DATA_BLOCK "Asi_output"	// DB 81
VERSION : 0.1
  STRUCT
   Adres_1_bit_0 : BOOL ;	//Temporary placeholder variable
   Adres_1_bit_1 : BOOL ;
   Adres_1_bit_2 : BOOL ;
   Adres_1_bit_3 : BOOL ;
   Adres_0_bit_0 : BOOL ;	//Temporary placeholder variable
   Adres_0_bit_1 : BOOL ;
   Adres_0_bit_2 : BOOL ;
   Adres_0_bit_3 : BOOL ;
   Adres_3_bit_0 : BOOL ;	//Temporary placeholder variable
   Adres_3_bit_1 : BOOL ;
   Adres_3_bit_2 : BOOL ;
   Adres_3_bit_3 : BOOL ;
   Adres_2_bit_0 : BOOL ;	//Temporary placeholder variable
   Adres_2_bit_1 : BOOL ;
   Adres_2_bit_2 : BOOL ;
   Adres_2_bit_3 : BOOL ;
   Adres_5_bit_0 : BOOL ;	//Temporary placeholder variable
   Adres_5_bit_1 : BOOL ;
   Adres_5_bit_2 : BOOL ;
   Adres_5_bit_3 : BOOL ;
   Adres_4_bit_0 : BOOL ;	//Temporary placeholder variable
   Adres_4_bit_1 : BOOL ;
   Adres_4_bit_2 : BOOL ;
   Adres_4_bit_3 : BOOL ;
   Adres_7_bit_0 : BOOL ;	//Temporary placeholder variable
   Adres_7_bit_1 : BOOL ;
   Adres_7_bit_2 : BOOL ;
   Adres_7_bit_3 : BOOL ;
   Adres_6_bit_0 : BOOL ;	//Temporary placeholder variable
   Adres_6_bit_1 : BOOL ;
   Adres_6_bit_2 : BOOL ;
   Adres_6_bit_3 : BOOL ;
   Adres_9_bit_0 : BOOL ;	//Temporary placeholder variable
   Adres_9_bit_1 : BOOL ;
   Adres_9_bit_2 : BOOL ;
   Adres_9_bit_3 : BOOL ;
   Adres_8_bit_0 : BOOL ;	//Temporary placeholder variable
   Adres_8_bit_1 : BOOL ;
   Adres_8_bit_2 : BOOL ;
   Adres_8_bit_3 : BOOL ;
   Adres_11_bit_0 : BOOL ;	//Temporary placeholder variable
   Adres_11_bit_1 : BOOL ;
   Adres_11_bit_2 : BOOL ;
   Adres_11_bit_3 : BOOL ;
   Adres_10_bit_0 : BOOL ;	//Temporary placeholder variable
   Adres_10_bit_1 : BOOL ;
   Adres_10_bit_2 : BOOL ;
   Adres_10_bit_3 : BOOL ;
   Adres_13_bit_0 : BOOL ;	//Temporary placeholder variable
   Adres_13_bit_1 : BOOL ;
   Adres_13_bit_2 : BOOL ;
   Adres_13_bit_3 : BOOL ;
   Adres_12_bit_0 : BOOL ;	//Temporary placeholder variable
   Adres_12_bit_1 : BOOL ;
   Adres_12_bit_2 : BOOL ;
   Adres_12_bit_3 : BOOL ;
   Adres_15_bit_0 : BOOL ;	//Temporary placeholder variable
   Adres_15_bit_1 : BOOL ;
   Adres_15_bit_2 : BOOL ;
   Adres_15_bit_3 : BOOL ;
   Adres_14_bit_0 : BOOL ;	//Temporary placeholder variable
   Adres_14_bit_1 : BOOL ;
   Adres_14_bit_2 : BOOL ;
   Adres_14_bit_3 : BOOL ;
   Adres_17_bit_0 : BOOL ;	//Temporary placeholder variable
   Adres_17_bit_1 : BOOL ;
   Adres_17_bit_2 : BOOL ;
   Adres_17_bit_3 : BOOL ;
   Adres_16_bit_0 : BOOL ;	//Temporary placeholder variable
   Adres_16_bit_1 : BOOL ;
   Adres_16_bit_2 : BOOL ;
   Adres_16_bit_3 : BOOL ;
   Adres_19_bit_0 : BOOL ;	//Temporary placeholder variable
   Adres_19_bit_1 : BOOL ;
   Adres_19_bit_2 : BOOL ;
   Adres_19_bit_3 : BOOL ;
   Adres_18_bit_0 : BOOL ;	//Temporary placeholder variable
   Adres_18_bit_1 : BOOL ;
   Adres_18_bit_2 : BOOL ;
   Adres_18_bit_3 : BOOL ;
   Adres_21_bit_0 : BOOL ;	//Temporary placeholder variable
   Adres_21_bit_1 : BOOL ;
   Adres_21_bit_2 : BOOL ;
   Adres_21_bit_3 : BOOL ;
   Adres_20_bit_0 : BOOL ;	//Temporary placeholder variable
   Adres_20_bit_1 : BOOL ;
   Adres_20_bit_2 : BOOL ;
   Adres_20_bit_3 : BOOL ;
   Adres_23_bit_0 : BOOL ;	//Temporary placeholder variable
   Adres_23_bit_1 : BOOL ;
   Adres_23_bit_2 : BOOL ;
   Adres_23_bit_3 : BOOL ;
   Adres_22_bit_0 : BOOL ;	//Temporary placeholder variable
   Adres_22_bit_1 : BOOL ;
   Adres_22_bit_2 : BOOL ;
   Adres_22_bit_3 : BOOL ;
   Adres_25_bit_0 : BOOL ;	//Temporary placeholder variable
   Adres_25_bit_1 : BOOL ;
   Adres_25_bit_2 : BOOL ;
   Adres_25_bit_3 : BOOL ;
   Adres_24_bit_0 : BOOL ;	//Temporary placeholder variable
   Adres_24_bit_1 : BOOL ;
   Adres_24_bit_2 : BOOL ;
   Adres_24_bit_3 : BOOL ;
   Adres_27_bit_0 : BOOL ;	//Temporary placeholder variable
   Adres_27_bit_1 : BOOL ;
   Adres_27_bit_2 : BOOL ;
   Adres_27_bit_3 : BOOL ;
   Adres_26_bit_0 : BOOL ;	//Temporary placeholder variable
   Adres_26_bit_1 : BOOL ;
   Adres_26_bit_2 : BOOL ;
   Adres_26_bit_3 : BOOL ;
   Adres_29_bit_0 : BOOL ;	//Temporary placeholder variable
   Adres_29_bit_1 : BOOL ;
   Adres_29_bit_2 : BOOL ;
   Adres_29_bit_3 : BOOL ;
   Adres_28_bit_0 : BOOL ;	//Temporary placeholder variable
   Adres_28_bit_1 : BOOL ;
   Adres_28_bit_2 : BOOL ;
   Adres_28_bit_3 : BOOL ;
   Adres_31_bit_0 : BOOL ;	//Temporary placeholder variable
   Adres_31_bit_1 : BOOL ;
   Adres_31_bit_2 : BOOL ;
   Adres_31_bit_3 : BOOL ;
   Adres_30_bit_0 : BOOL ;	//Temporary placeholder variable
   Adres_30_bit_1 : BOOL ;
   Adres_30_bit_2 : BOOL ;
   Adres_30_bit_3 : BOOL ;
   B_Adres_1_bit_0 : BOOL ;	//Temporary placeholder variable
   B_Adres_1_bit_1 : BOOL ;
   B_Adres_1_bit_2 : BOOL ;
   B_Adres_1_bit_3 : BOOL ;
   B_Adres_0_bit_0 : BOOL ;
   B_Adres_0_bit_1 : BOOL ;
   B_Adres_0_bit_2 : BOOL ;
   B_Adres_0_bit_3 : BOOL ;
   B_Adres_3_bit_0 : BOOL ;	//Temporary placeholder variable
   B_Adres_3_bit_1 : BOOL ;
   B_Adres_3_bit_2 : BOOL ;
   B_Adres_3_bit_3 : BOOL ;
   B_Adres_2_bit_0 : BOOL ;	//Temporary placeholder variable
   B_Adres_2_bit_1 : BOOL ;
   B_Adres_2_bit_2 : BOOL ;
   B_Adres_2_bit_3 : BOOL ;
   B_Adres_5_bit_0 : BOOL ;	//Temporary placeholder variable
   B_Adres_5_bit_1 : BOOL ;
   B_Adres_5_bit_2 : BOOL ;
   B_Adres_5_bit_3 : BOOL ;
   B_Adres_4_bit_0 : BOOL ;	//Temporary placeholder variable
   B_Adres_4_bit_1 : BOOL ;
   B_Adres_4_bit_2 : BOOL ;
   B_Adres_4_bit_3 : BOOL ;
   B_Adres_7_bit_0 : BOOL ;	//Temporary placeholder variable
   B_Adres_7_bit_1 : BOOL ;
   B_Adres_7_bit_2 : BOOL ;
   B_Adres_7_bit_3 : BOOL ;
   B_Adres_6_bit_0 : BOOL ;	//Temporary placeholder variable
   B_Adres_6_bit_1 : BOOL ;
   B_Adres_6_bit_2 : BOOL ;
   B_Adres_6_bit_3 : BOOL ;
   B_Adres_9_bit_0 : BOOL ;	//Temporary placeholder variable
   B_Adres_9_bit_1 : BOOL ;
   B_Adres_9_bit_2 : BOOL ;
   B_Adres_9_bit_3 : BOOL ;
   B_Adres_8_bit_0 : BOOL ;	//Temporary placeholder variable
   B_Adres_8_bit_1 : BOOL ;
   B_Adres_8_bit_2 : BOOL ;
   B_Adres_8_bit_3 : BOOL ;
   B_Adres_11_bit_0 : BOOL ;	//Temporary placeholder variable
   B_Adres_11_bit_1 : BOOL ;
   B_Adres_11_bit_2 : BOOL ;
   B_Adres_11_bit_3 : BOOL ;
   B_Adres_10_bit_0 : BOOL ;	//Temporary placeholder variable
   B_Adres_10_bit_1 : BOOL ;
   B_Adres_10_bit_2 : BOOL ;
   B_Adres_10_bit_3 : BOOL ;
   B_Adres_13_bit_0 : BOOL ;	//Temporary placeholder variable
   B_Adres_13_bit_1 : BOOL ;
   B_Adres_13_bit_2 : BOOL ;
   B_Adres_13_bit_3 : BOOL ;
   B_Adres_12_bit_0 : BOOL ;	//Temporary placeholder variable
   B_Adres_12_bit_1 : BOOL ;
   B_Adres_12_bit_2 : BOOL ;
   B_Adres_12_bit_3 : BOOL ;
   B_Adres_15_bit_0 : BOOL ;	//Temporary placeholder variable
   B_Adres_15_bit_1 : BOOL ;
   B_Adres_15_bit_2 : BOOL ;
   B_Adres_15_bit_3 : BOOL ;
   B_Adres_14_bit_0 : BOOL ;	//Temporary placeholder variable
   B_Adres_14_bit_1 : BOOL ;
   B_Adres_14_bit_2 : BOOL ;
   B_Adres_14_bit_3 : BOOL ;
   B_Adres_17_bit_0 : BOOL ;	//Temporary placeholder variable
   B_Adres_17_bit_1 : BOOL ;
   B_Adres_17_bit_2 : BOOL ;
   B_Adres_17_bit_3 : BOOL ;
   B_Adres_16_bit_0 : BOOL ;	//Temporary placeholder variable
   B_Adres_16_bit_1 : BOOL ;
   B_Adres_16_bit_2 : BOOL ;
   B_Adres_16_bit_3 : BOOL ;
   B_Adres_19_bit_0 : BOOL ;	//Temporary placeholder variable
   B_Adres_19_bit_1 : BOOL ;
   B_Adres_19_bit_2 : BOOL ;
   B_Adres_19_bit_3 : BOOL ;
   B_Adres_18_bit_0 : BOOL ;	//Temporary placeholder variable
   B_Adres_18_bit_1 : BOOL ;
   B_Adres_18_bit_2 : BOOL ;
   B_Adres_18_bit_3 : BOOL ;
   B_Adres_21_bit_0 : BOOL ;	//Temporary placeholder variable
   B_Adres_21_bit_1 : BOOL ;
   B_Adres_21_bit_2 : BOOL ;
   B_Adres_21_bit_3 : BOOL ;
   B_Adres_20_bit_0 : BOOL ;	//Temporary placeholder variable
   B_Adres_20_bit_1 : BOOL ;
   B_Adres_20_bit_2 : BOOL ;
   B_Adres_20_bit_3 : BOOL ;
   B_Adres_23_bit_0 : BOOL ;	//Temporary placeholder variable
   B_Adres_23_bit_1 : BOOL ;
   B_Adres_23_bit_2 : BOOL ;
   B_Adres_23_bit_3 : BOOL ;
   B_Adres_22_bit_0 : BOOL ;	//Temporary placeholder variable
   B_Adres_22_bit_1 : BOOL ;
   B_Adres_22_bit_2 : BOOL ;
   B_Adres_22_bit_3 : BOOL ;
   B_Adres_25_bit_0 : BOOL ;	//Temporary placeholder variable
   B_Adres_25_bit_1 : BOOL ;
   B_Adres_25_bit_2 : BOOL ;
   B_Adres_25_bit_3 : BOOL ;
   B_Adres_24_bit_0 : BOOL ;	//Temporary placeholder variable
   B_Adres_24_bit_1 : BOOL ;
   B_Adres_24_bit_2 : BOOL ;
   B_Adres_24_bit_3 : BOOL ;
   B_Adres_27_bit_0 : BOOL ;	//Temporary placeholder variable
   B_Adres_27_bit_1 : BOOL ;
   B_Adres_27_bit_2 : BOOL ;
   B_Adres_27_bit_3 : BOOL ;
   B_Adres_26_bit_0 : BOOL ;	//Temporary placeholder variable
   B_Adres_26_bit_1 : BOOL ;
   B_Adres_26_bit_2 : BOOL ;
   B_Adres_26_bit_3 : BOOL ;
   B_Adres_29_bit_0 : BOOL ;	//Temporary placeholder variable
   B_Adres_29_bit_1 : BOOL ;
   B_Adres_29_bit_2 : BOOL ;
   B_Adres_29_bit_3 : BOOL ;
   B_Adres_28_bit_0 : BOOL ;	//Temporary placeholder variable
   B_Adres_28_bit_1 : BOOL ;
   B_Adres_28_bit_2 : BOOL ;
   B_Adres_28_bit_3 : BOOL ;
   B_Adres_31_bit_0 : BOOL ;	//Temporary placeholder variable
   B_Adres_31_bit_1 : BOOL ;
   B_Adres_31_bit_2 : BOOL ;
   B_Adres_31_bit_3 : BOOL ;
   B_Adres_30_bit_0 : BOOL ;	//Temporary placeholder variable
   B_Adres_30_bit_1 : BOOL ;
   B_Adres_30_bit_2 : BOOL ;
   B_Adres_30_bit_3 : BOOL ;
  END_STRUCT ;	
BEGIN
END_DATA_BLOCK

DATA_BLOCK "MPI_GD"	// DB 100
VERSION : 0.1
  STRUCT
   IN : STRUCT
    Life_Bit_Foliarka : BOOL ;
    Foliarka_Automatyka : BOOL ;
    Foliarka_Reczny : BOOL ;
    Foto_Banda_1 : BOOL ;
    Foto_Owijarka : BOOL ;
    Rezerwa_1 : BOOL ;
    Motor_10_Lewo : BOOL ;
    Motor_10_Prawo : BOOL ;
    Motor_11_Lewo : BOOL ;
    Motor_11_Prawo : BOOL ;
    Zezwolenie_Na_Wjazd_10 : BOOL ;
    Potw_Dost_Na_Wjazd_10 : BOOL ;
    Zabierz_Na_Bande_11 : BOOL ;
    Paleta_Obecna_Na_7_Tr : BOOL ;
    Help_INT : INT ;
   END_STRUCT ;
   OUT : STRUCT
    Life_Bit_Szafa : BOOL ;
    Szafa_Automatyka : BOOL ;
    Foto_1_Banda_10 : BOOL ;
    Foto_2_Banda_10 : BOOL ;
    Foto_Banda_11 : BOOL ;
    Silnik_10_OK : BOOL ;
    Silnik_11_OK : BOOL ;
    Zabierz_Na_Bande_10 : BOOL ;
    Zezwolenie_Na_Wyjazd_11 : BOOL ;
    Potw_Dost_Na_Wyjazd_11 : BOOL ;
    Obrot_Na_Poz_Wlot_1 : BOOL ;
    Zmien_Program_Na_4 : BOOL ;
    Zmien_Pragram_Na_3 : BOOL ;
    Foto_Banda_9 : BOOL ;
    Help_INT : INT ;
   END_STRUCT ;
  END_STRUCT ;	
BEGIN
END_DATA_BLOCK

DATA_BLOCK "Blok_Bledow"	// DB 119
VERSION : 0.1
  STRUCT
   Blad_Silnika_Adr_1 : BOOL ;	//Blad silnika o adresie 1 - rolki obrotnica bindownicy
   Blad_Silnika_Adr_2 : BOOL ;	//Blad silnika o adresie 2 - rolki wylot bindownicy
   Blad_Silnika_Adr_3 : BOOL ;	//Blad silnika o adresie 3 - rolki
   Blad_Silnika_Adr_4 : BOOL ;	//Blad silnika o adresie 4 - rolki
   Blad_Silnika_Adr_5 : BOOL ;	//Blad silnika o adresie 5 - rolki
   Blad_Silnika_Adr_6 : BOOL ;	//Blad silnika o adresie 6 - rolki
   Blad_Silnika_Adr_7 : BOOL ;	//Blad silnika o adresie 7 - rolki
   Blad_Silnika_Adr_8 : BOOL ;	//Blad silnika o adresie 8 - rolki
   Blad_Silnika_Adr_9 : BOOL ;	//Blad silnika o adresie 9 - rolki
   Blad_Silnika_Adr_10 : BOOL ;	//Blad silnika o adresie 10 - rolki
   Blad_Silnika_Adr_11 : BOOL ;	//Blad silnika o adresie 11 - rolki
   Blad_Silnika_Adr_12 : BOOL ;	//Blad silnika o adresie 12 - rolki
   Blad_Silnika_Adr_13 : BOOL ;	//Blad silnika o adresie 13 - rolki
   Blad_Silnika_Adr_14 : BOOL ;	//Blad silnika o adresie 14 - rolki
   Blad_Silnika_Adr_15 : BOOL ;	//Blad silnika o adresie 15 - silnik obrotnicy bindownicy
   Blad_Rygla_Adr_16 : BOOL ;	//Blad rygla drzwi o adresie 16
   Blad_Silnika_Adr_18 : BOOL ;	//Blad silnika o adresie 18 - silnik obrotnicy wyboru wlotu
   Blad_Silnika_Adr_20 : BOOL ;	//Blad silnika o adresie 20 - silnik obrotnicy etykietownicy
   Blad_Silnika_Adr_23 : BOOL ;	//Blad silnika o adresie 23 - rolki
   Blad_Silnika_Adr_24 : BOOL ;	//Blad silnika o adresie 24 - rolki
   Blad_Kurtyny_Adr_25 : BOOL ;	//Blad kurtyny wlotowej  adres 25
   Blad_Kurtyny_Adr_26 : BOOL ;	//Blad kurtyny wylotowej aders 26
   Blad_Not_Aus_27 : BOOL ;	//Blad Not Aus adres 27 - Not Aus szafa
   Blad_Not_Aus_28 : BOOL ;	//Blad Not Aus adres 28 - Not Aus poczatek lini
   Blad_Not_Aus_29 : BOOL ;	//Blad Not Aus adres 29 - Not Aus srodek lini
   Blad_Not_Aus_30 : BOOL ;	//Blad Not Aus adres 30 - Not Aus koniec lini
   Blad_Not_Aus_31 : BOOL ;	//Blad Not Aus adres 31 - Not Aus panel bindownicy
   Blad_Przek_Bezp_Bind : BOOL ;	//Strefa bezpieczenstwa rejonu bindownicy  niepotwierdzona(wejscie -I4.4)
   Ostrz_Bind_Blad : BOOL ;	//Blad ogolny bindownicy
   Ostrz_Bind_Nie_Cofnieta : BOOL ;	//Bindownica nie jest cofnieta
   Ostrz_Bind_Sygn_Bezp : BOOL ;	//Bindownica brak sygnalu bezpieczenstwa
   Ostrz_Bind_Nie_Jest_Auto : BOOL ;	//Bindownica nie jest w trybie automatycznym (wejscie -I2.4)
   Ostrz_Stol_Obr_Foto : BOOL ;	//Blad fotokomorek stolu obrotowego
   Ostrz_Obr_Stol_Obr_Pozyc : BOOL ;	//Stol obrotowy nie jest w pozycji 0
   Ostrz_Pokr_Foto_Tas_1 : BOOL ;	//Niewlasciwe Pokrycie fotkomorek na tasmie 1 (Przejedz do przodu w recznym )
   Ostrz_Pokr_Foto_Tas_2 : BOOL ;	//Niewlasciwe Pokrycie fotkomorek na tasmie 2 (Przejedz do przodu w recznym )
   Ostrz_Pokr_Foto_Obr : BOOL ;	//Niewlasciwe Pokrycie fotkomorek na obrotnicy (Przejedz do przodu w recznym )
   Ostrz_Pokr_Foto_Tas_4 : BOOL ;	//Niewlasciwe Pokrycie fotkomorek na tasmie 4 (Przejedz do przodu w recznym )
   Blad_Krok_1 : BOOL ;	//Blad kroku nr 1 (Przekrokczony czas jazdy  na zadana pozycje)
   Blad_Krok_2 : BOOL ;	//Blad kroku nr 2 (Przekrokczony czas szukania srodka palety)
   Blad_Krok_3 : BOOL ;	//Blad kroku nr 3 (Przekrokczony czas pozycjonowania palety lewo/prawo)
   Blad_Krok_4 : BOOL ;	//Blad kroku nr 4 (Przekrokczony czas strzalu bindownicy)
   Blad_Krok_5 : BOOL ;	//Blad kroku nr 5 (Przekrokczony czas czasu postoju)
   Blad_Krok_6 : BOOL ;	//Blad kroku nr 6 (Przekrokczony czas powrotu lewo/prawo)
   Alarm_Obr_Stol_Obr_Pozyc : BOOL ;	//Stol obrotowy nie jest w pozycji 0
   Alarm_Bind_Nie_Cofinieta : BOOL ;	//Bindownica nie cofnieta lub brak zezwolenia  (cofnij ramie do tylu)
   Alarm_Bind_Sygn_Bezp : BOOL ;	//Bindownica brak sygnalu bezpieczenstwa
   rez3 : BOOL ;	//rez 3
   rez_6_0 : BOOL ;	//rez_6_0
   Alarm_Pokr_Foto_Tas_1 : BOOL ;	//Niewlasciwe Pokrycie fotkomorek na tasmie 1 (Przejedz do przodu w recznym )
   Alarm_Pokr_Foto_Tas_2 : BOOL ;	//Niewlasciwe Pokrycie fotkomorek na tasmie 2 (Przejedz do przodu w recznym )
   Alarm_Pokr_Foto_Tas_4 : BOOL ;	//Niewlasciwe Pokrycie fotkomorek na tasmie 4 (Przejedz do przodu w recznym )
   Alarm_Pokr_Foto_Obr : BOOL ;	//Niewlasciwe Pokrycie fotkomorek na obrotnicy przy braku cyklu
   Alarm_Bind_Nie_Jest_Auto : BOOL ;	//Bindownica nie jest w trybie automatycznym (wejscie -I2.4)
   Alarm_Bind_Blad : BOOL ;	//Blad ogolny bindownicy
   rez_6_7 : BOOL ;	//rez_6_7
   Ostrz_Prasa_Nie_W_Gorze : BOOL ;	//Zlamywak dekli nie jest u gory I2.6
   rez_7_1 : BOOL ;	//rez_7_1
   rez_7_2 : BOOL ;	//rez_7_2
   rez_7_3 : BOOL ;	//rez_7_3
   rez_7_4 : BOOL ;	//rez_7_4
   rez_7_5 : BOOL ;	//rez_7_5
   Ostrz_Wozek_Przy_Przen : BOOL ;	//Wozek widlowy przy przenosniku (i2.7)
   Ostrz_C_Bind_Foto_Pokr : BOOL ;	//Pokrycie fotokomorek podczas cyklu bindowania
   Ostrz_C_Bind_Poz_Bindow : BOOL ;	//Pozycja bindownicy podczas bindowania
   rez_8_1 : BOOL ;	//rez_8_1
   rez_8_2 : BOOL ;	//rez_8_2
   rez_8_3 : BOOL ;	//rez_8_3
   rez_8_4 : BOOL ;	//rez_8_4
   rez_8_5 : BOOL ;	//rez_8_5
   rez_8_6 : BOOL ;	//rez_8_6
   rez_8_7 : BOOL ;	//rez_8_7
   rez_9_0 : BOOL ;	//rez_9_0
   rez_9_1 : BOOL ;	//rez_9_1
   rez_9_2 : BOOL ;	//rez_9_2
   rez_9_3 : BOOL ;	//rez_9_3
   rez_9_4 : BOOL ;	//rez_9_4
   rez_9_5 : BOOL ;	//rez_9_5
   rez_9_6 : BOOL ;	//rez_9_6
   rez_9_7 : BOOL ;	//rez_9_7
   rez_int_bl : INT ;
   rez_int_bl_2 : INT ;
  END_STRUCT ;	
BEGIN
END_DATA_BLOCK

DATA_BLOCK "DB_HMI"	// DB 120
VERSION : 0.1
  STRUCT
   HMI_IN : STRUCT 	//Zmienne wchodzace do HMI nie nadpisywane W HMI (100 bajtow)
    Tryb_Reczny : BOOL ;	//Tryb Reczny
    Tryb_Auto : BOOL ;	//Tryb Auto
    Pozycja_0_st : BOOL ;	//Obrotnica Pozycja 0 st
    Pozycja_90_st : BOOL ;	//Obrotnica Pozycja 90 st
    Pozycja_180_st : BOOL ;	//Obrotnica Pozycja 180 st
    Pozycja_270_st : BOOL ;	//Obrotnica Pozycja 270 st
    Foto_Tasma_1_Tyl : BOOL ;	//foto tylne na bandzie wlotowej
    Foto_Tasma_1_Przod : BOOL ;	//foto przednie bandzie wlotowej
    Foto_Tasma_2_Tyl : BOOL ;	//foto tylne na bandzie wlotowej 2
    Foto_Tasma_2_Przod : BOOL ;	//foto przednie na bandzie wlotowej 2
    Foto_Obrotnica_3_Tyl : BOOL ;	//foto tylne na obrotnicy 3
    Foto_Obrotnica_3_Przod : BOOL ;	//foto przednie na obrotnicy 3
    Foto_Tasma_4_Tyl : BOOL ;	//foto tylne na bandzie wylotowej 4
    Foto_Tasma_4_Przod : BOOL ;	//foto przednie na bandzie wlotowej 4
    Motor_Tasma_1_Tyl : BOOL ;	//motor tasma 1 tyl
    Motor_Tasma_1_Przod : BOOL ;	//motor tasma 1 przod
    Motor_Tasma_2_Tyl : BOOL ;	//motor tasma 2 tyl
    Motor_Tasma_2_Przod : BOOL ;	//motor tasma 2 przod
    Motor_Tasma_3_Tyl : BOOL ;	//motor tasma obrotnica 3 tyl
    Motor_Tasma_3_Przod : BOOL ;	//motor tasma obrotnica 3 przod
    Motor_Obrotnica_3_CW : BOOL ;	//motor obrotnica 3 clock wise
    Motor_Obrotnica_3_CCW : BOOL ;	//motor obrotnica 3 counter clock wise
    Motor_Tasma_4_Przod : BOOL ;	//motor tasma obrotnica 4 tyl
    Motor_Tasma_4_Tyl : BOOL ;	//motor tasma obrotnica 4 przod
    Kurtyna_Wlot_Ok : BOOL ;	//kurtyna na wlocie ok
    Kurtyna_Wylot_Ok : BOOL ;	//kurtyna na wylocie ok
    Wybrano_TP_Przelot : BOOL ;	//wybrano tryb pracy przelot
    Wybrano_TP_Wiazanie_Wzdl : BOOL ;	//wybrano tryb pracy wiazanie wzdluzne
    Wybrano_TP_Wiazanie_Pop : BOOL ;	//wybrano tryb pracy wiazanie poprzeczne
    Wybrano_TP_Wiazanie_Krzy : BOOL ;	//wybrano tryb pracy wiazanie krzyzowe
    Czujnik_Ham_0_St : BOOL ;	//fotokomorka hamowania obrotnicy do kata 0st
    Czujnik_0_St : BOOL ;	//fotokomorka zatrzymania obrotnicy przy kacie 0st
    Czujnik_Ham_90_St : BOOL ;	//fotokomorka hamowania obrotnicy do kata 90st
    Czujnik_90_St : BOOL ;	//fotokomorka zatrzymania obrotnicy przy kacie 90st
    Czujnik_Ham_180_St : BOOL ;	//fotokomorka hamowania obrotnicy do kata 180st
    Czujnik_180_St : BOOL ;	//fotokomorka zatrzymania obrotnicy przy kacie 180st
    Czujnik_Ham_270_St : BOOL ;	//fotokomorka hamowania obrotnicy do kata 270st
    Czujnik_270_St : BOOL ;	//fotokomorka zatrzymania obrotnicy przy kacie 270st
    Interfefs_B_do_TP_B1 : BOOL ;	//obwod bezpieczenstwa bindownicy
    Interfefs_B_do_TP_B2 : BOOL ;	//polozenie podstawowe bindownicy
    Interfefs_B_do_TP_B3 : BOOL ;	//start/zakonczenie wiazania
    Interfefs_B_do_TP_B5 : BOOL ;	//blad bindownicy
    Interfefs_TP_do_B_TP1 : BOOL ;	//obwod bezpieczenstwa tasmociagow
    Interfefs_TP_do_B_TP2 : BOOL ;	//zezwolenie na prace bindownicy
    Interfefs_TP_do_B_TP3 : BOOL ;	//start wiazania
    PB_Strefa_bezpieczenstwa : BOOL ;	//przycisk zalaczenie Strefy bezpieczenstwa
    PB_Reczny : BOOL ;	//przycisk trybu reczny
    PB_Auto : BOOL ;	//przycisk auto
    PB_Reset : BOOL ;	//przycisk reset
    PB_Stop : BOOL ;	//przycisk stop
    PB_Cykl_Start : BOOL ;	//przycisk start cyklu
    PB_Tasma1_Tyl : BOOL ;	//przycisk tasma 1 do tylu
    PB_Tasma1_Przod : BOOL ;	//przycisk tasma 1 do przodu
    PB_Tasma2_Tyl : BOOL ;	//przycisk tasma 2 do tylu
    PB_Tasma2_Przod : BOOL ;	//przycisk tasma 2 do przodu
    PB_Tasma3_Tyl : BOOL ;	//przycisk tasma 3 do tylu
    PB_Tasma3_Przod : BOOL ;	//przycisk tasma 3 do przodu
    PB_Tasma4_Tyl : BOOL ;	//przycisk tasma 4 do tylu
    PB_Tasma4_Przod : BOOL ;	//przycisk tasma 4 do przodu
    PB_Tasma3_Obr_CW : BOOL ;	//przycisk obrotnica w prawo
    PB_Tasma3_Obr_CCW : BOOL ;	//przycisk obrotnica w lewo
    Lampka_Blad_Bind : BOOL ;	//lamka bledu bindownicy
    Lampka_Strzal_Tasmy : BOOL ;	//lampka wystrzalu tasmy
    Lampka_Strefa_Bezp : BOOL ;	//lampka przycisku strefy bezpieczenstwa
    Lampka_PB_Reczny : BOOL ;	//lampka przycisku trybu recznego
    Lampka_PB_Auto : BOOL ;	//lampka przycisku trybu auto
    Lampka_PB_Reset : BOOL ;	//lampka przycisku reset
    Lampka_PB_Stop : BOOL ;	//lampka przycisku stop
    Lampka_PB_Cykl_Start : BOOL ;	//lampka przycisku start
    Paleta_na_Tasmie_1 : BOOL ;	//znacznik palety na tasmie 1
    Paleta_na_Tasmie_2 : BOOL ;	//znacznik palety na tasmie 2
    Paleta_na_Tasmie_3_0_180 : BOOL ;	//znacznik palety na tasmie 3 przy kacie 0 lub 180st
    Paleta_na_Tasmie_3_90_27 : BOOL ;	//znacznik palety na tasmie 3 przy kacie 90 lub 270st
    Paleta_na_Tasmie_4 : BOOL ;	//znacznik palety na tasmie 4
    Paleta_na_Tasmie_1_T : BOOL ;	//znacznik palety na tasmie 1 wjazd
    Paleta_na_Tasmie_1_P : BOOL ;	//znacznik palety na tasmie 1 wyjazd
    Paleta_na_Tasmie_2_T : BOOL ;	//znacznik palety na tasmie 2 wjazd
    Paleta_na_Tasmie_2_P : BOOL ;	//znacznik palety na tasmie 2 wyjazd
    Paleta_na_Tasmie_3_T : BOOL ;	//znacznik palety na tasmie 3 wjazd
    Paleta_na_Tasmie_3_P : BOOL ;	//znacznik palety na tasmie 3 wyjazd
    Paleta_na_Tasmie_4_T : BOOL ;	//znacznik palety na tasmie 4 wjazd
    Paleta_na_Tasmie_4_P : BOOL ;	//znacznik palety na tasmie 4 wyjazd
    Rygiel : BOOL ;	//znacznik rygla drzwi
    Blad : BOOL ;	//Znacznik bledu
    Linia_transportowa_praca : BOOL ;	//Znacznik pracy calej linii transportowej
    Interfefs_B_do_TP_B4 : BOOL ;	//tryb pracy bindownicy: Auto(1) Reczny(0)
    Krok_1 : BOOL ;	//krok 1 trybu pracy
    Krok_2 : BOOL ;	//krok 2 trybu pracy
    Krok_3 : BOOL ;	//krok 3 trybu pracy
    Krok_4 : BOOL ;	//krok 4 trybu pracy
    Krok_5 : BOOL ;	//krok 5 trybu pracy
    Krok_6 : BOOL ;	//krok 6 trybu pracy
    Znacznik_Migania_Bledu : BOOL ;	//znacznik migania bledu
    Czujnik_Prasa : BOOL ;	//czujnik prasy s 22
    Stan_Zaworu : BOOL ;
    Tablica_IN_bool : ARRAY  [1 .. 10 ] OF BOOL  := FALSE;
    Tablica_IN_Byte : ARRAY  [1 .. 6 ] OF BYTE  := B#16#0;
    input_0 : BYTE ;
    input_1 : BYTE ;
    input_2 : BYTE ;
    input_3 : BYTE ;
    output_0 : BYTE ;
    output_1 : BYTE ;
    output_2 : BYTE ;
    output_3 : BYTE ;
    input_8 : BYTE ;
    input_9 : BYTE ;
    input_10 : BYTE ;
    input_11 : BYTE ;
    Tablica_IN_DWORD : ARRAY  [1 .. 4 ] OF DWORD ;
    NR_Kroku : DINT ;	//Numer kroku
    Aktualna_Data : DATE_AND_TIME ;
    Tablica_IN_INT : ARRAY  [1 .. 18 ] OF INT ;
    tryb_wiaz : INT ;	//znacznik wyboru trybu wiazania
    INT_Liczba_Akt_Kroku : INT ;	//znacznik wyboru aktualnie wykonywanego kroku
   END_STRUCT ;
   HMI_OUT : STRUCT 	//Zmienne wychodzace z HMI Nie nadpisywane w sterowniku od 100 bajta
    Rezerwa_Out_1 : BOOL ;
    Rezerwa_Out_2 : BOOL ;
    Start_Lini_z_OP : BOOL ;	//start calej lini z HMI
    Stop_Lini_z_OP : BOOL ;	//stop calej lini z HMI
    Wyzwolenie_Wyjazdu : BOOL ;	//wyzwolenie wyjazdu palety na stanowisku bindujacym (tylko w auto)
    Przycisk_Test_Lampek : BOOL ;	//przycisk test lampek
    Przycisk_Reset_Bledow : BOOL ;	//Przycisk resetowania bledow na panelu HMI
    Przycisk_Pozycjonowanie : BOOL ;	//Przycisk HMI do pozycjonowania palety
    H_Zalacz_Zawor_Prasa : BOOL ;	//Zalacz zawor prasa
    H_Zezwl_Ekran_Prasa : BOOL ;	//Zezwolenie na prase reczny
    Tablica_OUT_Bool : ARRAY  [1 .. 144 ] OF BOOL ;
    Tablina_OUT_INT : ARRAY  [1 .. 40 ] OF INT ;
   END_STRUCT ;
   HMI_IN_OUT : STRUCT 	//Zmienne nadpisywane w sterowniku i w HMI od 200 bajta
    Rezerwa_IN_Out_1 : BOOL ;
    Tp_Przelot : BOOL ;	//Tryb Pracy Przelot
    Tp_Wiazanie_Poprzeczne : BOOL ;	//Tryb Pracy Wiazanie poprzeczne
    Tp_Wiazanie_Wzdluzne : BOOL ;	//Tryb Pracy Wiazanie wzduzne
    Tp_Wiazanie_Pop_Wzdl : BOOL ;	//Tryb Pracy Wiaznie Poprzeczne i wzdluzne
    Tp_Pozycjonowanie : BOOL ;	//Tryb Pracy Pozycjonowanie Palety zalaczone
    Test_Lampek : BOOL ;	//Test Lampek
    Reset_bledow : BOOL ;	//Reset Bledow
    Zlamywak_Dekl : BOOL ;	//lamanie dekli
    Tablica_IN_OUT_Bool : ARRAY  [1 .. 144 ] OF BOOL ;
    Tablica_IN_OUT_INT : ARRAY  [1 .. 40 ] OF INT ;
    Wybor_trybu_pracy : BYTE ;
   END_STRUCT ;
  END_STRUCT ;	
BEGIN
   HMI_IN.Foto_Obrotnica_3_Przod := TRUE;
END_DATA_BLOCK

DATA_BLOCK DB 200
VERSION : 0.1
  STRUCT
   Wiazanie_Wzdluzne : BOOL ;	//wiazanie wzdluz palety
   Wiazanie_Poprzeczne : BOOL ;	//wiaznaie w poprzek palety
   Czas_Kontr_Rolki_Wlot : TIME  := T#12S;	//czas kontrolny wlotu
   Czas_Dojazd_Rolki_Wlot : TIME  := T#100MS;	//czas dojazdu do fotokomorki
   Czas_Opoz_Opusz_Bandy : TIME  := T#2S;	//czas po ktorym paleta opuszcza bande
   Czas_Opusz_Bandy : TIME  := T#2S;
   Czas_Opoz_Po_Strzale : TIME  := T#2S;
   Pozycjonowanie : BOOL ;	//jezeli true paleta pozycjonowana
   Pozycj_0_Lewo : BOOL ;	//pozycjonowanie 0st
   Pozycj_0_Prawo : BOOL ;	//pozycjonowanie 0st
   Pozycj_180_Lewo : BOOL ;	//pozycjonowanie 180st
   Pozycjo_180_Prawo : BOOL ;	//pozycjonowanie 180st
   Pozycj_0_Lewo_Czas : TIME  := T#2S;	//pozycjonowanie w lewo czas
   Pozycj_0_Prawo_Czas : TIME  := T#2S;	//pozycjonowanie w prawo czas
   Pozycj_180_Lewo_Czas : TIME  := T#2S;	//pozycjonowanie w lewo czas
   Pozycj_180_Prawo_Czas : TIME  := T#2S;	//pozycjonowanie w lewo czas
  END_STRUCT ;	
BEGIN
   Czas_Kontr_Rolki_Wlot := T#12S;
   Czas_Dojazd_Rolki_Wlot := T#100MS;
   Czas_Opoz_Opusz_Bandy := T#2S;
   Czas_Opusz_Bandy := T#2S;
   Czas_Opoz_Po_Strzale := T#2S;
   Pozycj_0_Lewo_Czas := T#2S;
   Pozycj_0_Prawo_Czas := T#2S;
   Pozycj_180_Lewo_Czas := T#2S;
   Pozycj_180_Prawo_Czas := T#2S;
END_DATA_BLOCK

ORGANIZATION_BLOCK OB 1
TITLE = "Main Program Sweep (Cycle)"
VERSION : 0.1
VAR_TEMP
  OB1_EV_CLASS : BYTE ;	//Bits 0-3 = 1 (Coming event), Bits 4-7 = 1 (Event class 1)
  OB1_SCAN_1 : BYTE ;	//1 (Cold restart scan 1 of OB 1), 3 (Scan 2-n of OB 1)
  OB1_PRIORITY : BYTE ;	//Priority of OB Execution
  OB1_OB_NUMBR : BYTE ;	//1 (Organization block 1, OB1)
  OB1_RESERVED_1 : BYTE ;	//Reserved for system
  OB1_RESERVED_2 : BYTE ;	//Reserved for system
  OB1_PREV_CYCLE : INT ;	//Cycle time of previous OB1 scan (milliseconds)
  OB1_MIN_CYCLE : INT ;	//Minimum cycle time of OB1 (milliseconds)
  OB1_MAX_CYCLE : INT ;	//Maximum cycle time of OB1 (milliseconds)
  OB1_DATE_TIME : DATE_AND_TIME ;	//Date and time OB1 started
END_VAR
BEGIN
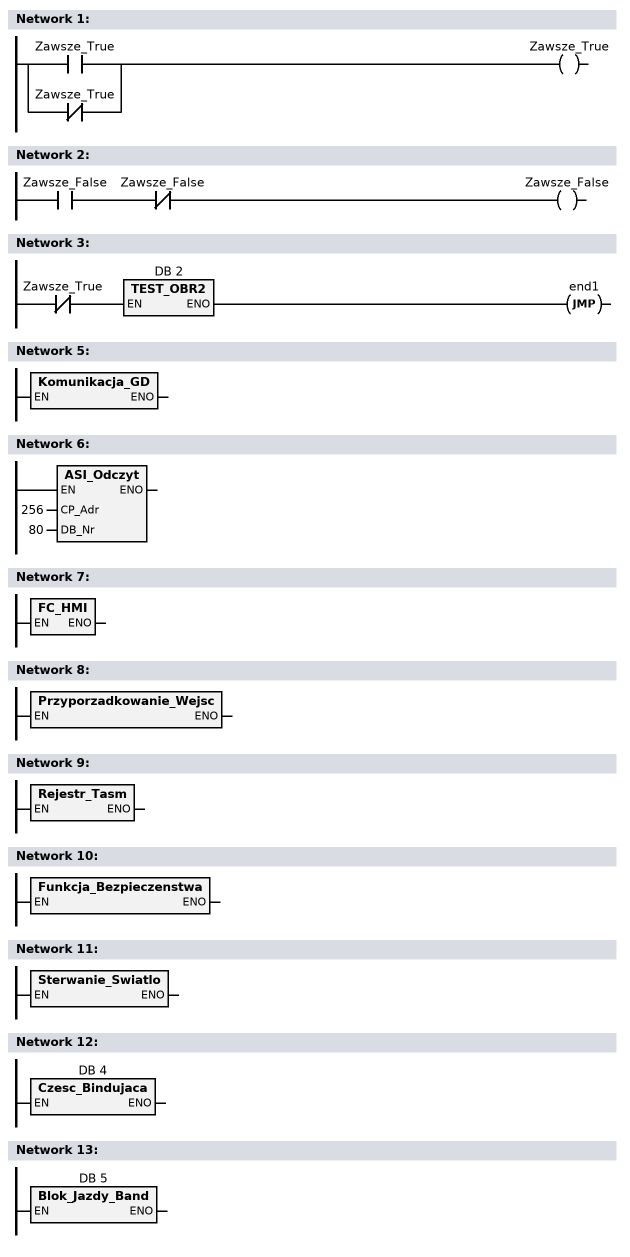
NETWORK
TITLE =
//Zawsze true
      O     "Zawsze_True";
      ON    "Zawsze_True";
      =     "Zawsze_True";
NETWORK
TITLE =
//Zawsze False
      A     "Zawsze_False";
      AN    "Zawsze_False";
      =     "Zawsze_False";
NETWORK
TITLE =
//Nie uzywany w normalej pracy blok
      AN    "Zawsze_True";
      JNB   _001;
      CALL  "TEST_OBR2" , DB 2;
_001: A     BR;
      JC    end1;
NETWORK
TITLE =
//to jest specjalny komentarz 
//do testow
//    BEU   
NETWORK
TITLE =
//   BEU   
      CALL  "Komunikacja_GD";
      NOP   0;
NETWORK
TITLE =
//Odczyt wejsc ASI
      CALL  "ASI_Odczyt" (
           CP_Adr                   := 256,
           DB_Nr                    := 80);
      NOP   0;
NETWORK
TITLE =
//komunikacja z hmi
      CALL  "FC_HMI";
      NOP   0;
NETWORK
TITLE =
      CALL  "Przyporzadkowanie_Wejsc";
      NOP   0;
NETWORK
TITLE =
      CALL  "Rejestr_Tasm";
      NOP   0;
NETWORK
TITLE =
      CALL  "Funkcja_Bezpieczenstwa";
      NOP   0;
NETWORK
TITLE =
      CALL  "Sterwanie_Swiatlo";
      NOP   0;
NETWORK
TITLE =
      CALL  "Czesc_Bindujaca" , DB 4;
      NOP   0;
NETWORK
TITLE =
      CALL  "Blok_Jazdy_Band" , DB 5;
      NOP   0;
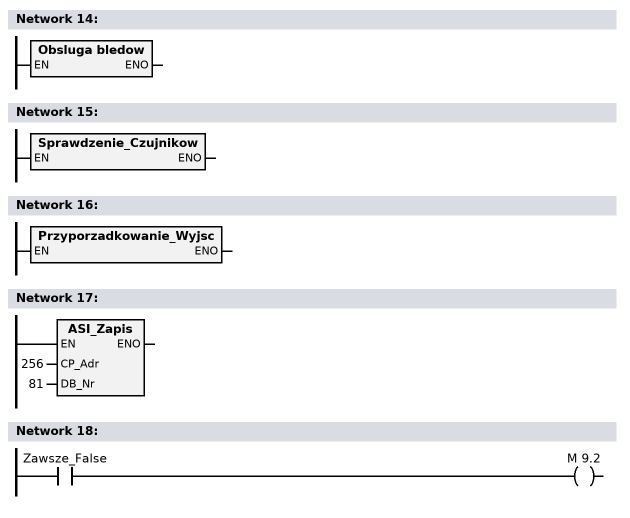
NETWORK
TITLE =
      CALL  "Obsluga bledow";
      NOP   0;
NETWORK
TITLE =
      CALL  "Sprawdzenie_Czujnikow";
      NOP   0;
NETWORK
TITLE =
      CALL  "Przyporzadkowanie_Wyjsc";
      NOP   0;
NETWORK
TITLE =
      CALL  "ASI_Zapis" (
           CP_Adr                   := 256,
           DB_Nr                    := 81);
      NOP   0;
NETWORK
TITLE =
end1: A     "Zawsze_False";
      =     M 9.2;
NETWORK
TITLE =
END_ORGANIZATION_BLOCK

ORGANIZATION_BLOCK "I/O_FLT1"	// OB 82
TITLE = "I/O Point Fault"
VERSION : 0.1
VAR_TEMP
  OB82_EV_CLASS : BYTE ;	//16#39, Event class 3, Entering event state, Internal fault event
  OB82_FLT_ID : BYTE ;	//16#XX, Fault identifcation code
  OB82_PRIORITY : BYTE ;	//Priority of OB Execution
  OB82_OB_NUMBR : BYTE ;	//82 (Organization block 82, OB82)
  OB82_RESERVED_1 : BYTE ;	//Reserved for system
  OB82_IO_FLAG : BYTE ;	//Input (01010100), Output (01010101)
  OB82_MDL_ADDR : WORD ;	//Base address of module with fault
  OB82_MDL_DEFECT : BOOL ;	//Module defective
  OB82_INT_FAULT : BOOL ;	//Internal fault
  OB82_EXT_FAULT : BOOL ;	//External fault
  OB82_PNT_INFO : BOOL ;	//Point information
  OB82_EXT_VOLTAGE : BOOL ;	//External voltage low
  OB82_FLD_CONNCTR : BOOL ;	//Field wiring connector missing
  OB82_NO_CONFIG : BOOL ;	//Module has no configuration data
  OB82_CONFIG_ERR : BOOL ;	//Module has configuration error
  OB82_MDL_TYPE : BYTE ;	//Type of module
  OB82_SUB_MDL_ERR : BOOL ;	//Sub-Module is missing or has error
  OB82_COMM_FAULT : BOOL ;	//Communication fault
  OB82_MDL_STOP : BOOL ;	//Module is stopped
  OB82_WTCH_DOG_FLT : BOOL ;	//Watch dog timer stopped module
  OB82_INT_PS_FLT : BOOL ;	//Internal power supply fault
  OB82_PRIM_BATT_FLT : BOOL ;	//Primary battery is in fault
  OB82_BCKUP_BATT_FLT : BOOL ;	//Backup battery is in fault
  OB82_RESERVED_2 : BOOL ;	//Reserved for system
  OB82_RACK_FLT : BOOL ;	//Rack fault, only for bus interface module
  OB82_PROC_FLT : BOOL ;	//Processor fault
  OB82_EPROM_FLT : BOOL ;	//EPROM fault
  OB82_RAM_FLT : BOOL ;	//RAM fault
  OB82_ADU_FLT : BOOL ;	//ADU fault
  OB82_FUSE_FLT : BOOL ;	//Fuse fault
  OB82_HW_INTR_FLT : BOOL ;	//Hardware interupt input in fault
  OB82_RESERVED_3 : BOOL ;	//Reserved for system
  OB82_DATE_TIME : DATE_AND_TIME ;	//Date and time OB82 started
END_VAR
BEGIN
NETWORK
TITLE =
END_ORGANIZATION_BLOCK

ORGANIZATION_BLOCK "RACK_FLT"	// OB 86
TITLE = "Loss Of Rack Fault"
VERSION : 0.1
VAR_TEMP
  OB86_EV_CLASS : BYTE ;	//16#38/39 Event class 3
  OB86_FLT_ID : BYTE ;	//16#C1/C4/C5, Fault identifcation code
  OB86_PRIORITY : BYTE ;	//Priority of OB Execution
  OB86_OB_NUMBR : BYTE ;	//86 (Organization block 86, OB86)
  OB86_RESERVED_1 : BYTE ;	//Reserved for system
  OB86_RESERVED_2 : BYTE ;	//Reserved for system
  OB86_MDL_ADDR : WORD ;	//Base address of IM module in rack with fault
  OB86_RACKS_FLTD : ARRAY  [0 .. 31 ] OF BOOL ;	//Racks in fault
  OB86_DATE_TIME : DATE_AND_TIME ;	//Date and time OB86 started
END_VAR
BEGIN
// (block stored without names or comments; labels and parameter names are numbered)
END_ORGANIZATION_BLOCK

ORGANIZATION_BLOCK "COMPLETE RESTART"	// OB 100
TITLE = "Complete Restart"
VERSION : 0.1
VAR_TEMP
  OB100_EV_CLASS : BYTE ;	//16#13, Event class 1, Entering event state, Event logged in diagnostic buffer
  OB100_STRTUP : BYTE ;	//16#81/82/83/84 Method of startup
  OB100_PRIORITY : BYTE ;	//Priority of OB Execution
  OB100_OB_NUMBR : BYTE ;	//100 (Organization block 100, OB100)
  OB100_RESERVED_1 : BYTE ;	//Reserved for system
  OB100_RESERVED_2 : BYTE ;	//Reserved for system
  OB100_STOP : WORD ;	//Event that caused CPU to stop (16#4xxx)
  OB100_STRT_INFO : DWORD ;	//Information on how system started
  OB100_DATE_TIME : DATE_AND_TIME ;	//Date and time OB100 started
END_VAR
BEGIN
NETWORK
TITLE =
END_ORGANIZATION_BLOCK

ORGANIZATION_BLOCK "PROG_ERR"	// OB 121
TITLE = "Programming Error"
VERSION : 0.1
VAR_TEMP
  OB121_EV_CLASS : BYTE ;	//16#25, Event class 2, Entering event state, Internal fault event
  OB121_SW_FLT : BYTE ;	//16#XX Software programming fault
  OB121_PRIORITY : BYTE ;	//Priority of OB Execution
  OB121_OB_NUMBR : BYTE ;	//121 (Organization block 121, OB121)
  OB121_BLK_TYPE : BYTE ;	//16#88/8A/8B/8C/8E Type of block fault occured in
  OB121_RESERVED_1 : BYTE ;	//Reserved for system
  OB121_FLT_REG : WORD ;	//16#XX Specific register that caused fault
  OB121_BLK_NUM : WORD ;	//Number of block that programming fault occured in
  OB121_PRG_ADDR : WORD ;	//Address in block where programming fault occured
  OB121_DATE_TIME : DATE_AND_TIME ;	//Date and time OB121 started
END_VAR
BEGIN
NETWORK
TITLE =
END_ORGANIZATION_BLOCK

SYMBOL_TABLE
"AIO"	DB 10	DB 10
"Blok_Para"	DB 12	DB 12
"Blok_Bledow_Program"	DB 13	DB 13
"Asi_input"	DB 80	DB 80
"Asi_output"	DB 81	DB 81
"MPI_GD"	DB 100	DB 100	// Blok wymiany danych po mpi
"Blok_Bledow"	DB 119	DB 119
"DB_HMI"	DB 120	DB 120	// Blok wejsc wyjsc HMI
"Czesc_Bindujaca"	FB 3	FB 3	// Blok jazdy band bindownicy
"Czesc_Trasnportujaca"	FB 5	FB 5
"T_ON"	FB 20	FB 20	// Timer on delay with memory
"T_ON_+_RESET"	FB 21	FB 21	// Czasowka on delay z zapamietanym czasem  + reset
"Banda_Pojedyncza"	FB 30	FB 30
"Banda_Obr_1"	FB 31	FB 31	// Banda obrotowa o dwoch wlotach i jednej fotokomorce
"Banda_Obr_2"	FB 32	FB 32	// Banda obrotowa nr 2
"Banda_Poj_+Tryb_Reczny"	FB 33	FB 33
"Banda_Obr_Bind"	FB 34	FB 34	// Banda obrotowa sluzaca do bindowania
"Blok_Pracy_Bindownicy"	FB 35	FB 35	// funkcja pozycjonujaca bande
"Wybranie_Wjazdu"	FB 50	FB 50
"Obr_Na_Poz_1"	FB 51	FB 51
"Obr_Na_Poz_2"	FB 52	FB 52	// Obrot na pozycje uwzgledniajacy czujniki 45st
"Obr_Na_Poz_4"	FB 54	FB 54
"Pozycjonowanie_Bandy"	FB 55	FB 55
"Bindownica_Test"	FB 57	FB 57	// Testowy blok wejsc wyjsc bindownicy
"Pozycjonowanie_Palety"	FB 58	FB 58	// Funkcja pozycjonujaca palete
"Funkcja_Bezpieczenstwa"	FC 3	FC 3
"Sprawdzenie_Czujnikow"	FC 4	FC 4
"FC_Lampki"	FC 6	FC 6	// Funkcja sterujaca lampkami
"Szukaj_Zmiany_2"	FC 7	FC 7
"Toggle"	FC 8	FC 8	// Funkcja przycisku bistabilnego
"Sterwanie_Swiatlo"	FC 9	FC 9	// Sterowanie sygnalami swietlnymi
"Przyporzadkowanie_Wejsc"	FC 20	FC 20
"Przyporzadkowanie_Wyjsc"	FC 21	FC 21
"Rejestr_Tasm"	FC 30	FC 30
"FC_Auto_Reczny"	FC 40	FC 40
"Przycisk_Reset"	FC 41	FC 41	// Kasowanie_Bledow
"ASI_Odczyt"	FC 80	FC 80
"ASI_Zapis"	FC 81	FC 81
"Opoznienie_Wylotu"	FC 85	FC 85
"Opoznienie_Wlotu"	FC 86	FC 86	// Funkcja opozniajaca wlot
"Komunikacja_GD"	FC 100	FC 100	// Komunikacja szafa foliarka
"Obsluga bledow"	FC 119	FC 119	// funkcja przekazujaca bledy do bloku db
"FC_HMI"	FC 120	FC 120
"Funkcja_Zegara"	FC 140	FC 140	// Funkcja zegara
"I/O_FLT1"	OB 82	OB 82	// I/O Point Fault 1
"RACK_FLT"	OB 86	OB 86	// Loss of Rack Fault
"COMPLETE RESTART"	OB 100	OB 100	// Complete Restart
"PROG_ERR"	OB 121	OB 121	// Programming Error
"TON"	SFB 4	SFB 4	// Generate an On Delay
"READ_CLK"	SFC 1	SFC 1	// Read System Clock
"WR_REC"	SFC 58	SFC 58	// Write Data Record
"RD_REC"	SFC 59	SFC 59	// Read a Data Record
"SEW_Model"	UDT 1	UDT 1	// Model SEW'a
"CROSS_Model"	UDT 2	UDT 2
"ESTOP_Model"	UDT 3	UDT 3
"PB_Model"	UDT 5	UDT 5	// Model przycisku
"OBROTOWA_Model"	UDT 6	UDT 6	// Model sygnalow z bandy obrotowej
"CZUJNIKI_1_Model"	UDT 7	UDT 7	// Model czujnikow na obrotnicy
"CZUJNIKI_2_Model"	UDT 8	UDT 8
"S_Model"	UDT 9	UDT 9
"CZUJNIKI_3_MODEL"	UDT 10	UDT 10
"OBROTOWA_2_MODEL"	UDT 11	UDT 11
"RESET_MODEL"	UDT 12	UDT 12
"Wzor_Pracy"	UDT 20	UDT 20
"VAT_1"	VAT 1	
"VAT3"	VAT 3	
"VAT4"	VAT 4	
"VAT_Para"	VAT 5	
END_SYMBOL_TABLE

TYPE "SEW_Model"	// UDT 1
VERSION : 0.1
  STRUCT
   Silnik_OK : BOOL ;	//Silnik ok
   Rezerwa_Silnik : BOOL ;
   Foto_1 : BOOL ;	//Wejscie SEW 1
   Foto_2 : BOOL ;	//Wejscie SEW 2
   C_Wise : BOOL ;	//ClockWise
   CC_Wise : BOOL ;	//CounterClockWise
   Wolno : BOOL ;	//Wolno
   S_Bit : BOOL ;	//Bit bezpieczenstwa
   Zez_Do_Pop : BOOL ;	//Zezwolenie do poprzedniej
   Paleta_Dost_do_Pop : BOOL ;	//Potwierdzenie dostarczenia
   Zabierz_do_Nast : BOOL ;	//Przejecie palety do nast
   Paleta_Poprawna : BOOL ;	//Wykorzystywane do monitoringu
   Res_1_4 : BOOL ;
   Res_1_5 : BOOL ;
   Zez_Reczny_do_Pop : BOOL ;	//Zezwolenie na reczny tyl
   Zez_Reczny_do_Nast : BOOL ;	//Zezwolenie na reczny przod
  END_STRUCT ;	
END_TYPE

TYPE "CROSS_Model"	// UDT 2
VERSION : 0.1
  STRUCT
   OSSD_Tor_1_1 : BOOL ;
   OSSD_Tor_1_2 : BOOL ;
   OSSD_Tor_2_1 : BOOL ;
   OSSD_Tor_2_2 : BOOL ;
   Rez_0_4 : BOOL ;
   Rez_0_5 : BOOL ;
   Rez_0_6 : BOOL ;
   Rez_0_7 : BOOL ;
   Rez_1_0 : BOOL ;
   Rez_1_1 : BOOL ;
   Rez_1_2 : BOOL ;
   Rez_1_3 : BOOL ;
   Rez_1_4 : BOOL ;
   Rez_1_5 : BOOL ;
   Rez_1_6 : BOOL ;
   Rez_1_7 : BOOL ;
  END_STRUCT ;	
END_TYPE

TYPE "ESTOP_Model"	// UDT 3
VERSION : 0.1
  STRUCT
   EStop_Tor_1_1 : BOOL ;
   EStop_Tor_1_2 : BOOL ;
   EStop_Tor_2_1 : BOOL ;
   EStop_Tor_2_2 : BOOL ;
   Rez_0_4 : BOOL ;
   Rez_0_5 : BOOL ;
   Rez_0_6 : BOOL ;
   Rez_0_7 : BOOL ;
   Rez_1_0 : BOOL ;
   Rez_1_1 : BOOL ;
   Rez_1_2 : BOOL ;
   Rez_1_3 : BOOL ;
   Rez_1_4 : BOOL ;
   Rez_1_5 : BOOL ;
   Rez_1_6 : BOOL ;
   Rez_1_7 : BOOL ;
  END_STRUCT ;	
END_TYPE

TYPE "PB_Model"	// UDT 5
VERSION : 0.1
  STRUCT
   Przycisk_Start : BOOL ;	//Start i reset ob. bezp
   Czujnik_Kolizji : BOOL ;
   Rez_0_2 : BOOL ;
   Rez_0_3 : BOOL ;
   Rez_0_4 : BOOL ;
   Rez_0_5 : BOOL ;
   Rez_0_6 : BOOL ;
   Rez_0_7 : BOOL ;
   Rez_1_0 : BOOL ;
   Rez_1_1 : BOOL ;
   Rez_1_2 : BOOL ;
   Rez_1_3 : BOOL ;
   Rez_1_4 : BOOL ;
   Rez_1_5 : BOOL ;
   Rez_1_6 : BOOL ;
   Rez_1_7 : BOOL ;
  END_STRUCT ;	
END_TYPE

TYPE "OBROTOWA_Model"	// UDT 6
VERSION : 0.1
  STRUCT
   Silnik_OK : BOOL ;	//Silnik ok
   Rezerwa_Silnik : BOOL ;
   Foto_1 : BOOL ;	//Wejscie SEW 1
   Foto_2 : BOOL ;	//Wejscie SEW 2
   C_Wise : BOOL ;	//ClockWise
   CC_Wise : BOOL ;	//CounterClockWise
   Wolno : BOOL ;	//Wolno
   S_Bit : BOOL ;	//Bit bezpieczenstwa
   Zez_Do_Pop_Wlot_1 : BOOL ;	//Zezwolenie do poprzedniej
   Potw_Dost_Wlot_1 : BOOL ;	//Potwierdzenie dostarczenia
   Zez_Do_Pop_Wlot_2 : BOOL ;	//Wykorzystywane do monitoringu
   Potw_Dost_Wlot_2 : BOOL ;
   Przejmij_Palete : BOOL ;	//Przejecie palety do nast
   Rez_1_6 : BOOL ;
   Paleta_Poprawna_1 : BOOL ;	//Wykorzystywane do monitoringu
  END_STRUCT ;	
END_TYPE

TYPE "CZUJNIKI_1_Model"	// UDT 7
VERSION : 0.1
  STRUCT
   Czujnik_0_St : BOOL ;
   Czujnik_Ham_0_St : BOOL ;
   Czujnik_Ham_90_St : BOOL ;
   Czujnik_90_St : BOOL ;
   Rez_0_4 : BOOL ;
   Rez_0_5 : BOOL ;
   Rez_0_6 : BOOL ;
   Rez_0_7 : BOOL ;
   Rez_1_0 : BOOL ;
   Rez_1_1 : BOOL ;
   Rez_1_2 : BOOL ;
   Rez_1_3 : BOOL ;
   Rez_1_4 : BOOL ;
   Rez_1_5 : BOOL ;
   Rez_1_6 : BOOL ;
   Rez_1_7 : BOOL ;
  END_STRUCT ;	
END_TYPE

TYPE "CZUJNIKI_2_Model"	// UDT 8
VERSION : 0.1
  STRUCT
   Czujnik_45_St_CW : BOOL ;
   Czujnik_45_St_CCW : BOOL ;
   Rez_0_2 : BOOL ;
   Rez_0_3 : BOOL ;
   Rez_0_4 : BOOL ;
   Rez_0_5 : BOOL ;
   Rez_0_6 : BOOL ;
   Rez_0_7 : BOOL ;
   Rez_1_0 : BOOL ;
   Rez_1_1 : BOOL ;
   Rez_1_2 : BOOL ;
   Rez_1_3 : BOOL ;
   Rez_1_4 : BOOL ;
   Rez_1_5 : BOOL ;
   Rez_1_6 : BOOL ;
   Rez_1_7 : BOOL ;
  END_STRUCT ;	
END_TYPE

TYPE "S_Model"	// UDT 9
VERSION : 0.1
  STRUCT
   Silnik_OK : BOOL ;	//Silnik ok
   Rezerwa_Silnik : BOOL ;
   Foto_1 : BOOL ;	//Wejscie SEW 1
   Foto_2 : BOOL ;	//Wejscie SEW 2
   C_Wise : BOOL ;	//ClockWise
   CC_Wise : BOOL ;	//CounterClockWise
   Wolno : BOOL ;	//Wolno
   S_Bit : BOOL ;	//Bit bezpieczenstwa
   Zez_Do_Pop_Wlot_1 : BOOL ;	//Zezwolenie do poprzedniej
   Potw_Dost_Wlot_1 : BOOL ;	//Potwierdzenie dostarczenia
   Zez_Do_Pop_Wlot_2 : BOOL ;	//Wykorzystywane do monitoringu
   Potw_Dost_Wlot_2 : BOOL ;
   Przejmij_Palete : BOOL ;	//Przejecie palety do nast
   Rez_1_6 : BOOL ;
   Paleta_Poprawna_1 : BOOL ;	//Wykorzystywane do monitoringu
  END_STRUCT ;	
END_TYPE

TYPE "CZUJNIKI_3_MODEL"	// UDT 10
VERSION : 0.1
  STRUCT
   Czujnik_Ham_180_St : BOOL ;
   Czujnik_180_St : BOOL ;
   Czujnik_Ham_270_St : BOOL ;
   Czujnik_270_St : BOOL ;
   Rez_0_4 : BOOL ;
   Rez_0_5 : BOOL ;
   Rez_0_6 : BOOL ;
   Rez_0_7 : BOOL ;
   Rez_1_0 : BOOL ;
   Rez_1_1 : BOOL ;
   Rez_1_2 : BOOL ;
   Rez_1_3 : BOOL ;
   Rez_1_4 : BOOL ;
   Rez_1_5 : BOOL ;
   Rez_1_6 : BOOL ;
   Rez_1_7 : BOOL ;
  END_STRUCT ;	
END_TYPE

TYPE "OBROTOWA_2_MODEL"	// UDT 11
VERSION : 0.1
  STRUCT
   Silnik_OK : BOOL ;	//Silnik ok
   Rezerwa_Silnik : BOOL ;
   Foto_1 : BOOL ;	//Wejscie SEW 1
   Foto_2 : BOOL ;	//Wejscie SEW 2
   C_Wise : BOOL ;	//ClockWise
   CC_Wise : BOOL ;	//CounterClockWise
   Wolno : BOOL ;	//Wolno
   S_Bit : BOOL ;	//Bit bezpieczenstwa
   Res_1_0 : BOOL ;	//Zezwolenie do poprzedniej
   Res_1_1 : BOOL ;	//Potwierdzenie dostarczenia
   Res_1_2 : BOOL ;	//Potwierdzenie dostarczenia
   Res_1_3 : BOOL ;	//Potwierdzenie dostarczenia
   Res_1_4 : BOOL ;	//Potwierdzenie dostarczenia
   Res_1_5 : BOOL ;	//Potwierdzenie dostarczenia
   Res_1_6 : BOOL ;	//Potwierdzenie dostarczenia
   Res_1_7 : BOOL ;	//Potwierdzenie dostarczenia
  END_STRUCT ;	
END_TYPE

TYPE "RESET_MODEL"	// UDT 12
VERSION : 0.1
  STRUCT
   Reset_Wlot : BOOL ;
   Reset_Wylot : BOOL ;
   RES_0_2 : BOOL ;
   RES_0_3 : BOOL ;
   Rez_0_4 : BOOL ;
   Rez_0_5 : BOOL ;
   Rez_0_6 : BOOL ;
   Rez_0_7 : BOOL ;
   Rez_1_0 : BOOL ;
   Rez_1_1 : BOOL ;
   Rez_1_2 : BOOL ;
   Rez_1_3 : BOOL ;
   Rez_1_4 : BOOL ;
   Rez_1_5 : BOOL ;
   Rez_1_6 : BOOL ;
   Rez_1_7 : BOOL ;
  END_STRUCT ;	
END_TYPE

TYPE "Wzor_Pracy"	// UDT 20
VERSION : 0.1
  STRUCT
   wiazanie_poprzeczne : BOOL ;
   wiazanie_wzdluzne : BOOL ;
  END_STRUCT ;	
END_TYPE

FUNCTION_BLOCK "Czesc_Bindujaca"	// FB 3
//Funkcja odpowiada za sterowanie lini bindujacej
//Uwzgledniony zostal tryb reczny
//
VERSION : 0.1
VAR
  Tasma_1 : FB 33;	//Adres 23
  Tasma_2 : FB 33;	//Adres 24
  Tasma_Obr_3 : FB 34;	//Adres 1 i 15
  Tasma_4 : FB 33;	//Adres 2
  Bin_IN_OUT : FB 57;
  Bind_Obwod_Ok : BOOL ;
  Bind_Poz_Podst : BOOL ;
  Bind_Sygn_Got : BOOL ;
  Bind_Blad : BOOL ;
  Bind_Start_Kon : BOOL ;
  Zaj_Nieb_2 : BOOL ;
  Zaj_Nieb_4 : BOOL ;
  Tasma_Rezerwa_1 : FB 33;
  Tasma_Rezerwa_2 : FB 33;
END_VAR
VAR_TEMP
  Temp_Bit_1 : BOOL ;
END_VAR
BEGIN
NETWORK
TITLE =
//Ten network celowo jest wolny
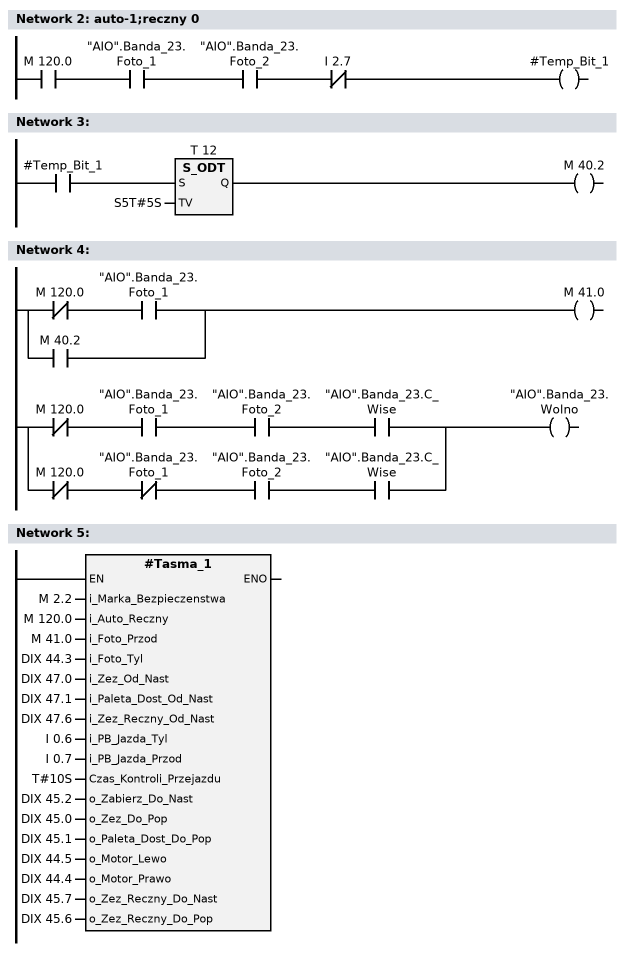
NETWORK
TITLE = auto-1;reczny 0
      A     M 120.0;
      A     "AIO".Banda_23.Foto_1;
      A     "AIO".Banda_23.Foto_2;
      AN    I 2.7;
      =     #Temp_Bit_1;
NETWORK
TITLE =
//Opoznienie startu po polozeniu palety
//
      A     #Temp_Bit_1;
      L     S5T#5S;
      SD    T 12;
      NOP   0;
      NOP   0;
      NOP   0;
      A     T 12;
      =     M 40.2;
NETWORK
TITLE =
//Opoznienie wlotu bandy 1
      AN    M 120.0;
      A     "AIO".Banda_23.Foto_1;
      O;
      A     M 40.2;
      =     M 41.0;
//Silnik wolno  aby nie spadl z bandy
      AN    M 120.0;
      A     "AIO".Banda_23.Foto_1;
      A     "AIO".Banda_23.Foto_2;
      A     "AIO".Banda_23.C_Wise;
//      A     "Zawsze_False"
      O;
      AN    M 120.0;
      AN    "AIO".Banda_23.Foto_1;
      A     "AIO".Banda_23.Foto_2;
      A     "AIO".Banda_23.C_Wise;
      =     "AIO".Banda_23.Wolno;
NETWORK
TITLE =
//Tasma 1 adres 23
      CALL  #Tasma_1 (
           i_Marka_Bezpieczenstwa   := M 2.2,
           i_Auto_Reczny            := M 120.0,
           i_Foto_Przod             := M 41.0,
           i_Foto_Tyl               := DIX 44.3,
           i_Zez_Od_Nast            := DIX 47.0,
           i_Paleta_Dost_Od_Nast    := DIX 47.1,
           i_Zez_Reczny_Od_Nast     := DIX 47.6,
           i_PB_Jazda_Tyl           := I 0.6,
           i_PB_Jazda_Przod         := I 0.7,
           Czas_Kontroli_Przejazdu  := T#10S,
           o_Zabierz_Do_Nast        := DIX 45.2,
           o_Zez_Do_Pop             := DIX 45.0,
           o_Paleta_Dost_Do_Pop     := DIX 45.1,
           o_Motor_Lewo             := DIX 44.5,
           o_Motor_Prawo            := DIX 44.4,
           o_Zez_Reczny_Do_Nast     := DIX 45.7,
           o_Zez_Reczny_Do_Pop      := DIX 45.6);	//kierunek normalny lini
      NOP   0;
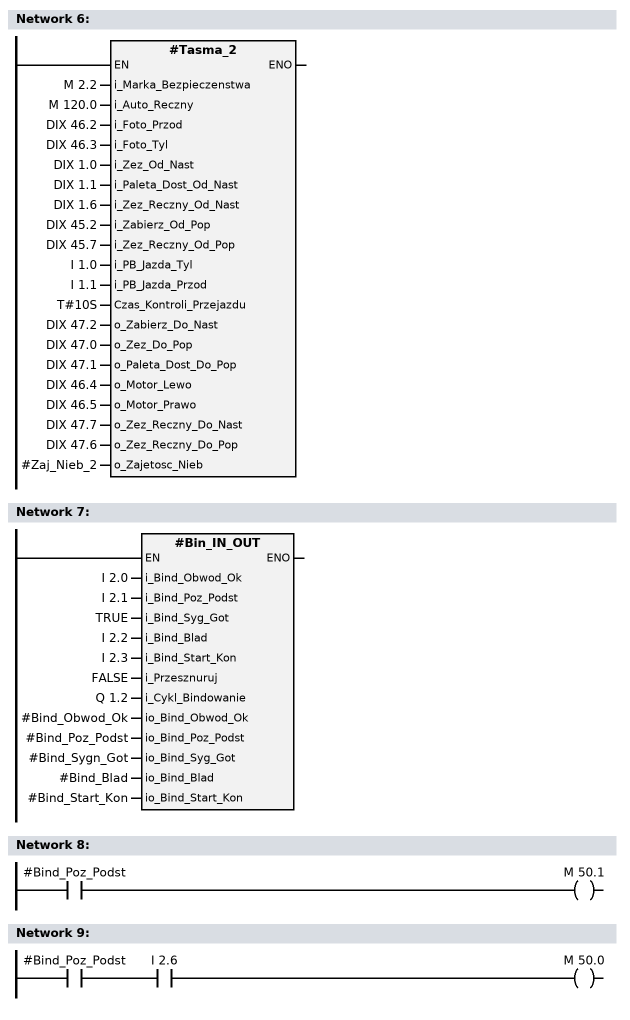
NETWORK
TITLE =
//Tasma 2 adres 24
      CALL  #Tasma_2 (
           i_Marka_Bezpieczenstwa   := M 2.2,
           i_Auto_Reczny            := M 120.0,
           i_Foto_Przod             := DIX 46.2,
           i_Foto_Tyl               := DIX 46.3,
           i_Zez_Od_Nast            := DIX 1.0,
           i_Paleta_Dost_Od_Nast    := DIX 1.1,
           i_Zez_Reczny_Od_Nast     := DIX 1.6,
           i_Zabierz_Od_Pop         := DIX 45.2,
           i_Zez_Reczny_Od_Pop      := DIX 45.7,
           i_PB_Jazda_Tyl           := I 1.0,
           i_PB_Jazda_Przod         := I 1.1,
           Czas_Kontroli_Przejazdu  := T#10S,
           o_Zabierz_Do_Nast        := DIX 47.2,
           o_Zez_Do_Pop             := DIX 47.0,
           o_Paleta_Dost_Do_Pop     := DIX 47.1,
           o_Motor_Lewo             := DIX 46.4,
           o_Motor_Prawo            := DIX 46.5,
           o_Zez_Reczny_Do_Nast     := DIX 47.7,
           o_Zez_Reczny_Do_Pop      := DIX 47.6,
           o_Zajetosc_Nieb          := #Zaj_Nieb_2);	//kierunek normalny lini
      NOP   0;
NETWORK
TITLE =
//blok przejsciowy  do bindownicy
//(maskuje sygnal wejscia i wyjscia)
      CALL  #Bin_IN_OUT (
           i_Bind_Obwod_Ok          := I 2.0,
           i_Bind_Poz_Podst         := I 2.1,
           i_Bind_Syg_Got           := TRUE,
           i_Bind_Blad              := I 2.2,
           i_Bind_Start_Kon         := I 2.3,
           i_Przesznuruj            := FALSE,
           i_Cykl_Bindowanie        := Q 1.2,
           io_Bind_Obwod_Ok         := #Bind_Obwod_Ok,
           io_Bind_Poz_Podst        := #Bind_Poz_Podst,
           io_Bind_Syg_Got          := #Bind_Sygn_Got,
           io_Bind_Blad             := #Bind_Blad,
           io_Bind_Start_Kon        := #Bind_Start_Kon);
NETWORK
TITLE =
      A     #Bind_Poz_Podst;
      =     M 50.1;
NETWORK
TITLE =
      A     #Bind_Poz_Podst;
      A     I 2.6;
      =     M 50.0;
NETWORK
TITLE =
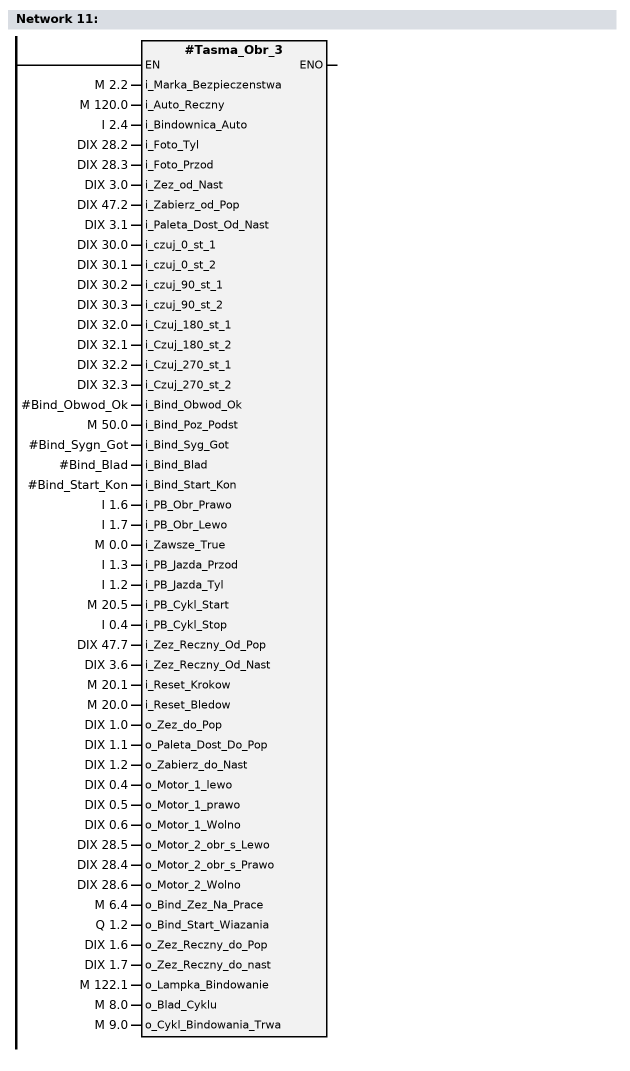
NETWORK
TITLE =
//bindownica z obrotnica
      CALL  #Tasma_Obr_3 (
           i_Marka_Bezpieczenstwa   := M 2.2,
           i_Auto_Reczny            := M 120.0,
           i_Bindownica_Auto        := I 2.4,
           i_Foto_Tyl               := DIX 28.2,
           i_Foto_Przod             := DIX 28.3,
           i_Zez_od_Nast            := DIX 3.0,
           i_Zabierz_od_Pop         := DIX 47.2,
           i_Paleta_Dost_Od_Nast    := DIX 3.1,
           i_czuj_0_st_1            := DIX 30.0,
           i_czuj_0_st_2            := DIX 30.1,
           i_czuj_90_st_1           := DIX 30.2,
           i_czuj_90_st_2           := DIX 30.3,
           i_Czuj_180_st_1          := DIX 32.0,
           i_Czuj_180_st_2          := DIX 32.1,
           i_Czuj_270_st_1          := DIX 32.2,
           i_Czuj_270_st_2          := DIX 32.3,
           i_Bind_Obwod_Ok          := #Bind_Obwod_Ok,
           i_Bind_Poz_Podst         := M 50.0,
           i_Bind_Syg_Got           := #Bind_Sygn_Got,
           i_Bind_Blad              := #Bind_Blad,
           i_Bind_Start_Kon         := #Bind_Start_Kon,
           i_PB_Obr_Prawo           := I 1.6,
           i_PB_Obr_Lewo            := I 1.7,
           i_Zawsze_True            := M 0.0,
           i_PB_Jazda_Przod         := I 1.3,
           i_PB_Jazda_Tyl           := I 1.2,
           i_PB_Cykl_Start          := M 20.5,
           i_PB_Cykl_Stop           := I 0.4,
           i_Zez_Reczny_Od_Pop      := DIX 47.7,
           i_Zez_Reczny_Od_Nast     := DIX 3.6,
           i_Reset_Krokow           := M 20.1,
           i_Reset_Bledow           := M 20.0,
           o_Zez_do_Pop             := DIX 1.0,
           o_Paleta_Dost_Do_Pop     := DIX 1.1,
           o_Zabierz_do_Nast        := DIX 1.2,
           o_Motor_1_lewo           := DIX 0.4,
           o_Motor_1_prawo          := DIX 0.5,
           o_Motor_1_Wolno          := DIX 0.6,
           o_Motor_2_obr_s_Lewo     := DIX 28.5,
           o_Motor_2_obr_s_Prawo    := DIX 28.4,
           o_Motor_2_Wolno          := DIX 28.6,
           o_Bind_Zez_Na_Prace      := M 6.4,
           o_Bind_Start_Wiazania    := Q 1.2,
           o_Zez_Reczny_do_Pop      := DIX 1.6,
           o_Zez_Reczny_do_nast     := DIX 1.7,
           o_Lampka_Bindowanie      := M 122.1,
           o_Blad_Cyklu             := M 8.0,
           o_Cykl_Bindowania_Trwa   := M 9.0);
NETWORK
TITLE = Zezwolenie na prase reczny
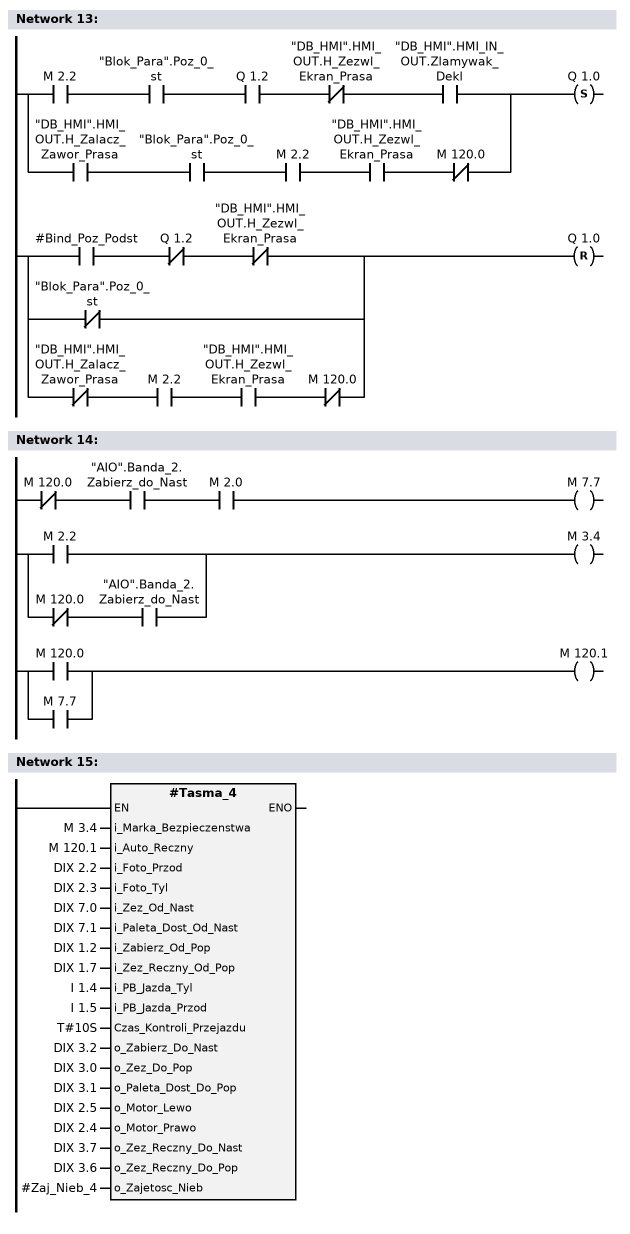
NETWORK
TITLE =
      A(;
      A     M 2.2;
      A     "Blok_Para".Poz_0_st;
      A     Q 1.2;
      AN    "DB_HMI".HMI_OUT.H_Zezwl_Ekran_Prasa;
      A     "DB_HMI".HMI_IN_OUT.Zlamywak_Dekl;
      O;
      A     "DB_HMI".HMI_OUT.H_Zalacz_Zawor_Prasa;
      A     "Blok_Para".Poz_0_st;
      A     M 2.2;
      A     "DB_HMI".HMI_OUT.H_Zezwl_Ekran_Prasa;
      AN    M 120.0;
      );
      S     Q 1.0;
      A(;
      A     #Bind_Poz_Podst;
      AN    Q 1.2;
      AN    "DB_HMI".HMI_OUT.H_Zezwl_Ekran_Prasa;
      ON    "Blok_Para".Poz_0_st;
      O;
      AN    "DB_HMI".HMI_OUT.H_Zalacz_Zawor_Prasa;
      A     M 2.2;
      A     "DB_HMI".HMI_OUT.H_Zezwl_Ekran_Prasa;
      AN    M 120.0;
      );
      R     Q 1.0;
      NOP   0;
NETWORK
TITLE =
//Nowa Marka bepieczenstwa na wyjazd
//Marka bepieczenstwa przejsciowa
      AN    M 120.0;
      A     "AIO".Banda_2.Zabierz_do_Nast;
      A     M 2.0;
      =     M 7.7;
      A     M 2.2;
      O;
      AN    M 120.0;
      A     "AIO".Banda_2.Zabierz_do_Nast;
      =     M 3.4;
//Jezeli marka bezpieczenstwa 3 auto zalaczone
      A     M 120.0;
      O;
      A     M 7.7;
      =     M 120.1;
NETWORK
TITLE =
//Tasma 4 adres 2
//Ta tasma pod wzgledem bezpieczenstwa nalezy do lini i bindownicy
//Nastepna banda jest obrotnica
//
//
//
      CALL  #Tasma_4 (
           i_Marka_Bezpieczenstwa   := M 3.4,
           i_Auto_Reczny            := M 120.1,
           i_Foto_Przod             := DIX 2.2,
           i_Foto_Tyl               := DIX 2.3,
           i_Zez_Od_Nast            := DIX 7.0,
           i_Paleta_Dost_Od_Nast    := DIX 7.1,
           i_Zabierz_Od_Pop         := DIX 1.2,
           i_Zez_Reczny_Od_Pop      := DIX 1.7,
           i_PB_Jazda_Tyl           := I 1.4,
           i_PB_Jazda_Przod         := I 1.5,
           Czas_Kontroli_Przejazdu  := T#10S,
           o_Zabierz_Do_Nast        := DIX 3.2,
           o_Zez_Do_Pop             := DIX 3.0,
           o_Paleta_Dost_Do_Pop     := DIX 3.1,
           o_Motor_Lewo             := DIX 2.5,
           o_Motor_Prawo            := DIX 2.4,
           o_Zez_Reczny_Do_Nast     := DIX 3.7,
           o_Zez_Reczny_Do_Pop      := DIX 3.6,
           o_Zajetosc_Nieb          := #Zaj_Nieb_4);	//kierunek normalny lini
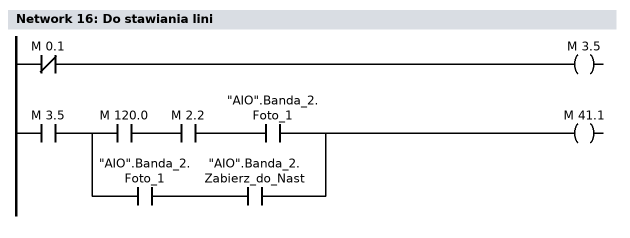
NETWORK
TITLE = Do stawiania lini
//Banda 2. Uznawana za Wlot 1
//Uwaga By dzialolo nalezy wymusic true
      AN    M 0.1;
      =     M 3.5;
//--
      A     M 3.5;
      A(;
      A     M 120.0;
      A     M 2.2;
      A     "AIO".Banda_2.Foto_1;
      O;
      A     "AIO".Banda_2.Foto_1;
      A     "AIO".Banda_2.Zabierz_do_Nast;
      );
      =     M 41.1;
END_FUNCTION_BLOCK

FUNCTION_BLOCK "Czesc_Trasnportujaca"	// FB 5
VERSION : 0.1
VAR
  Banda_1 : FB 30;
  Banda_2 : FB 30;
  Banda_3 : FB 30;
  Banda_4 : FB 31;
  Banda_5 : FB 30;
  Banda_6 : FB 30;
  Banda_7 : FB 30;
  Banda_8 : FB 30;
  Banda_9 : FB 30;
  Banda_12 : FB 30;
  Banda_13 : FB 32;
  Banda_14 : FB 30;
END_VAR
BEGIN
NETWORK
TITLE =
//Ten network celowo jest wolny
NETWORK
TITLE =
//Opoznienie wlotu bandy 1
//Uwaga Stare !!!
//      CALL  "Opoznienie_Wlotu"
//       Wejscie :="AIO".Banda_1.Foto_1
//       Timmer_1:=T12
//       Timmer_2:=T13
//       Wyjscie :="M_Foto_1_Banda_1"
//       Zmienna :="Help_M_40_3"
NETWORK
TITLE =
//Banda 1
//Uwaga Stare !!!
//      CALL  #Banda_1
//       S_Marka_Bezpieczenstwa :="Marka_Bezpieczenstwa"
//       i_Foto_Koniec          :="M_Foto_1_Banda_1"
//       i_Zez_Od_Nast          :="AIO".Banda_2.Zez_Do_Pop
//       i_Paleta_Dost_Od_Nast  :="AIO".Banda_2.Paleta_Dost_do_Pop
//       i_Zabierz_Od_Pop       :=
//       Czas_Kontroli_Przejazdu:=T#10S
//       o_Zabierz_Do_Nast      :="AIO".Banda_1.Zabierz_do_Nast
//       o_Zez_Do_Pop           :="AIO".Banda_1.Zez_Do_Pop
//       o_Paleta_Dost_do_Pop   :="AIO".Banda_1.Paleta_Dost_do_Pop
//       o_Motor_Lewo           :="AIO".Banda_1.C_Wise
NETWORK
TITLE =
//Banda 2. Uznawana za Wlot 1
//Uwaga Stare !!!
//      CALL  #Banda_2
//       S_Marka_Bezpieczenstwa :="Marka_Bezpieczenstwa"
//       i_Foto_Koniec          :="AIO".Banda_2.Foto_1
//       i_Zez_Od_Nast          :="AIO".Banda_4.Zez_Do_Pop_Wlot_1
//       i_Paleta_Dost_Od_Nast  :="AIO".Banda_4.Potw_Dost_Wlot_1
//       i_Zabierz_Od_Pop       :="AIO".Banda_1.Zabierz_do_Nast
//       Czas_Kontroli_Przejazdu:=T#10S
//       o_Zabierz_Do_Nast      :="AIO".Banda_2.Zabierz_do_Nast
//       o_Zez_Do_Pop           :="AIO".Banda_2.Zez_Do_Pop
//       o_Paleta_Dost_do_Pop   :="AIO".Banda_2.Paleta_Dost_do_Pop
//       o_Motor_Lewo           :="AIO".Banda_2.C_Wise
NETWORK
TITLE =
//Opoznienie wlotu banda 3
      CALL  "Opoznienie_Wlotu" (
           Wejscie                  := "AIO".Banda_3.Foto_1,
           Timmer_1                 := T 14,
           Timmer_2                 := T 15,
           Wyjscie                  := M 40.4,
           Zmienna                  := M 40.5);
NETWORK
TITLE =
//Banda 3. Uznawana za Wlot 2
      CALL  #Banda_3 (
           S_Marka_Bezpieczenstwa   := M 2.0,
           i_Foto_Koniec            := M 40.4,
           i_Zez_Od_Nast            := DIX 7.2,
           i_Paleta_Dost_Od_Nast    := DIX 7.3,
           Czas_Kontroli_Przejazdu  := T#10S,
           o_Zabierz_Do_Nast        := DIX 5.2,
           o_Zez_Do_Pop             := DIX 5.0,
           o_Paleta_Dost_do_Pop     := DIX 5.1,
           o_Motor_Lewo             := DIX 4.4);
NETWORK
TITLE =
//Banda 4 obrotowa
      CALL  #Banda_4 (
           i_Marka_bezpieczenstwa   := M 2.0,
           i_Foto_1                 := DIX 6.2,
           i_Foto_2                 := DIX 6.3,
           i_Zez_od_Nast            := DIX 9.0,
           i_Zabierz_od_Wlot_1      := DIX 3.2,
           i_Zabierz_od_Wlot_2      := DIX 5.2,
           i_Paleta_Odb_Wylot       := DIX 9.1,
           i_czuj_poz_Wlot_1        := DIX 36.3,
           i_czuj_ham_Wlot_1        := DIX 36.2,
           i_czuj_poz_Wlot_2        := DIX 36.0,
           i_czuj_ham_Wlot_2        := DIX 36.1,
           i_Foto_Wlot_1            := M 41.1,
           i_Foto_Wlot_2            := M 40.4,
           o_Zez_do_Wlot_1          := DIX 7.0,
           o_Zez_do_Wlot_2          := DIX 7.2,
           o_Paleta_Dost_Wlot_1     := DIX 7.1,
           o_Paleta_Dost_Wlot_2     := DIX 7.3,
           o_Zabierz_do_Nast        := DIX 7.4,
           o_Motor_1_lewo           := DIX 6.4,
           o_Motor_1_prawo          := DIX 6.5,
           o_Motor_2_obr_s_Wlot_1   := DIX 34.5,
           o_Motor_2_obr_s_Wlot_2   := DIX 34.4,
           o_Motor_2_Wolno          := DIX 34.6);
NETWORK
TITLE =
//Banda 5
      CALL  #Banda_5 (
           S_Marka_Bezpieczenstwa   := M 2.0,
           i_Foto_Koniec            := DIX 8.2,
           i_Zez_Od_Nast            := DIX 11.0,
           i_Paleta_Dost_Od_Nast    := DIX 11.1,
           i_Zabierz_Od_Pop         := DIX 7.4,
           Czas_Kontroli_Przejazdu  := T#10S,
           o_Zabierz_Do_Nast        := DIX 9.2,
           o_Zez_Do_Pop             := DIX 9.0,
           o_Paleta_Dost_do_Pop     := DIX 9.1,
           o_Motor_Lewo             := DIX 8.4);
NETWORK
TITLE =
//Banda 6
      CALL  #Banda_6 (
           S_Marka_Bezpieczenstwa   := M 2.0,
           i_Foto_Koniec            := DIX 10.2,
           i_Zez_Od_Nast            := DIX 13.0,
           i_Paleta_Dost_Od_Nast    := DIX 13.1,
           i_Zabierz_Od_Pop         := DIX 9.2,
           Czas_Kontroli_Przejazdu  := T#10S,
           o_Zabierz_Do_Nast        := DIX 11.2,
           o_Zez_Do_Pop             := DIX 11.0,
           o_Paleta_Dost_do_Pop     := DIX 11.1,
           o_Motor_Lewo             := DIX 10.4);
NETWORK
TITLE =
//Banda 7
      CALL  #Banda_7 (
           S_Marka_Bezpieczenstwa   := M 2.0,
           i_Foto_Koniec            := DIX 12.2,
           i_Zez_Od_Nast            := DIX 15.0,
           i_Paleta_Dost_Od_Nast    := DIX 15.1,
           i_Zabierz_Od_Pop         := DIX 11.2,
           Czas_Kontroli_Przejazdu  := T#10S,
           o_Zabierz_Do_Nast        := DIX 13.2,
           o_Zez_Do_Pop             := DIX 13.0,
           o_Paleta_Dost_do_Pop     := DIX 13.1,
           o_Motor_Lewo             := DIX 12.4);
NETWORK
TITLE =
//Banda 8
      CALL  #Banda_8 (
           S_Marka_Bezpieczenstwa   := M 2.0,
           i_Foto_Koniec            := DIX 14.2,
           i_Zez_Od_Nast            := DIX 17.0,
           i_Paleta_Dost_Od_Nast    := DIX 17.1,
           i_Zabierz_Od_Pop         := DIX 13.2,
           Czas_Kontroli_Przejazdu  := T#10S,
           o_Zabierz_Do_Nast        := DIX 15.2,
           o_Zez_Do_Pop             := DIX 15.0,
           o_Paleta_Dost_do_Pop     := DIX 15.1,
           o_Motor_Lewo             := DIX 14.4);
NETWORK
TITLE =
//Banda 9
      CALL  #Banda_9 (
           S_Marka_Bezpieczenstwa   := M 2.0,
           i_Foto_Koniec            := DIX 16.2,
           i_Zez_Od_Nast            := DIX 19.0,
           i_Paleta_Dost_Od_Nast    := DIX 19.1,
           i_Zabierz_Od_Pop         := DIX 15.2,
           Czas_Kontroli_Przejazdu  := T#10S,
           o_Zabierz_Do_Nast        := DIX 17.2,
           o_Zez_Do_Pop             := DIX 17.0,
           o_Paleta_Dost_do_Pop     := DIX 17.1,
           o_Motor_Lewo             := DIX 16.4);
NETWORK
TITLE = Zezwolenie do poprzedniej
//Banda 10 to foliarka. Tu jest interface laczacy dwie maszyny
      A     "MPI_GD".IN.Zezwolenie_Na_Wjazd_10;
      =     "AIO".Banda_10.Zez_Do_Pop;
//---
      A     "MPI_GD".IN.Potw_Dost_Na_Wjazd_10;
      =     "AIO".Banda_10.Paleta_Dost_do_Pop;
      A     "AIO".Banda_9.Zabierz_do_Nast;
      =     "MPI_GD".OUT.Zabierz_Na_Bande_10;
NETWORK
TITLE =
//Banda 11 to wylot z foliarki. Tu jest interface laczacy.Uwazana jako wlot 1
      A     "AIO".Banda_13.Zez_Do_Pop_Wlot_1;
      =     "MPI_GD".OUT.Zezwolenie_Na_Wyjazd_11;
//Przedluzenine czasu trwania sygnalu potwierdzenia
      A     "AIO".Banda_13.Potw_Dost_Wlot_1;
      L     S5T#200MS;
      SE    T 20;
      A     T 20;
      =     "MPI_GD".OUT.Potw_Dost_Na_Wyjazd_11;
//Przejecie palety
      A     "MPI_GD".IN.Zabierz_Na_Bande_11;
      =     "AIO".Banda_11.Zabierz_do_Nast;
      A     "MPI_GD".IN.Paleta_Obecna_Na_7_Tr;
      =     M 30.0;
      A     "AIO".Czuj_21.Czujnik_90_St;
      AN    "AIO".Czuj_21.Czujnik_0_St;
      AN    "AIO".Czuj_22.Czujnik_45_St_CW;
      AN    "AIO".Czuj_22.Czujnik_45_St_CCW;
      =     "MPI_GD".OUT.Obrot_Na_Poz_Wlot_1;
NETWORK
TITLE =
//Opoznienie wlotu 2 przy obrotnicy 2
      CALL  "Opoznienie_Wlotu" (
           Wejscie                  := "AIO".Banda_12.Foto_1,
           Timmer_1                 := T 16,
           Timmer_2                 := T 17,
           Wyjscie                  := M 40.6,
           Zmienna                  := M 40.7);
NETWORK
TITLE =
//Banda 12. Uwazana jako wlot 2.
      CALL  #Banda_12 (
           S_Marka_Bezpieczenstwa   := M 2.0,
           i_Foto_Koniec            := M 40.6,
           i_Zez_Od_Nast            := DIX 25.2,
           i_Paleta_Dost_Od_Nast    := DIX 25.3,
           Czas_Kontroli_Przejazdu  := T#10S,
           o_Zabierz_Do_Nast        := DIX 23.2,
           o_Zez_Do_Pop             := DIX 23.0,
           o_Paleta_Dost_do_Pop     := DIX 23.1,
           o_Motor_Lewo             := DIX 22.4);
NETWORK
TITLE =
//banda 13 obrotowa
      CALL  #Banda_13 (
           i_Marka_bezpieczenstwa   := M 2.0,
           i_Foto_1                 := DIX 24.2,
           i_Foto_2                 := DIX 24.3,
           i_Zez_od_Nast            := DIX 27.0,
           i_Zabierz_od_Wlot_1      := DIX 21.2,
           i_Zabierz_od_Wlot_2      := DIX 23.2,
           i_Paleta_Odb_Wylot       := DIX 27.1,
           i_czuj_poz_Wlot_1        := DIX 40.3,
           i_czuj_ham_Wlot_1        := DIX 40.2,
           i_czuj_poz_Wlot_2        := DIX 40.0,
           i_czuj_ham_Wlot_2        := DIX 40.1,
           i_Czuj_poz_45_deg        := DIX 42.0,
           i_Czuj_ham_45_deg        := DIX 42.1,
           i_Foto_Wlot_1            := M 30.0,
           i_Foto_Wlot_2            := M 40.6,
           i_Etyk_praca_wlacz       := I 4.3,
           i_Etyk_poz_podst         := I 5.0,
           i_Etyk_obraz_w_pamieci   := I 5.2,
           i_Etyk_syg_gotowosci     := I 5.1,
           i_Etyk_brak_materialu    := I 5.3,
           i_Etyk_Przycisk_Drukuj   := I 5.4,
           o_Zez_do_Wlot_1          := DIX 25.0,
           o_Zez_do_Wlot_2          := DIX 25.2,
           o_Paleta_Dost_Wlot_1     := DIX 25.1,
           o_Paleta_Dost_Wlot_2     := DIX 25.3,
           o_Zabierz_do_Nast        := DIX 25.4,
           o_Motor_1_lewo           := DIX 24.4,
           o_Motor_1_prawo          := DIX 24.5,
           o_Motor_2_obr_s_Wlot_1   := DIX 38.5,
           o_Motor_2_obr_s_Wlot_2   := DIX 38.4,
           o_Motor_2_Wolno          := DIX 38.6,
           o_Silownik_etykiety      := Q 8.4,
           o_Drukuj_Etykiete        := Q 8.5,
           o_Zalaczenie_Skanera     := Q 8.6,
           o_Lampka_Przycisk_Drukuj := Q 9.0);
NETWORK
TITLE =
//Wywolanie opoznienia zatrzymania fotokomorki po wyjsciu z obrotnicy
      CALL  "Opoznienie_Wylotu" (
           Wejscie                  := "AIO".Banda_14.Foto_1,
           Timmer_1                 := T 10,
           Timmer_2                 := T 11,
           Wyjscie                  := M 40.0,
           Zmienna                  := M 40.1);
NETWORK
TITLE =
//Banda 14.Banda uwazana jako wylot z obrotnicy.
      CALL  #Banda_14 (
           S_Marka_Bezpieczenstwa   := M 2.0,
           i_Foto_Koniec            := M 40.0,
           i_Zabierz_Od_Pop         := DIX 25.4,
           Czas_Kontroli_Przejazdu  := T#10S,
           o_Zabierz_Do_Nast        := DIX 27.2,
           o_Zez_Do_Pop             := DIX 27.0,
           o_Paleta_Dost_do_Pop     := DIX 27.1,
           o_Motor_Lewo             := DIX 26.4);
//      SET   
//      S     "Zalacz_Skaner"
END_FUNCTION_BLOCK

FUNCTION_BLOCK "T_ON"	// FB 20
//Funkcja zatrzymujaca czas gdy na wejsciu stop pojawi sie stan niski. Wartosc 
//wejscia TON nie jest wtedy brana pod uwage. 
AUTHOR : Kng
NAME : Help_FB
VERSION : 0.1
VAR_INPUT
  IN : BOOL ;	//Wejscie aktywujace timer
  STOP : BOOL ;	//Sygnal aktywny stanem wysokim
  PT : TIME ;	//Czas zadany
END_VAR
VAR_OUTPUT
  Q_0 : BOOL ;
END_VAR
VAR_IN_OUT
  ET : TIME ;
END_VAR
VAR
  T_1 : SFB 4;
  Help_Zbocze_1 : BOOL ;
  Help_Zbocze_2 : BOOL ;
  Help_Zbocze_3 : BOOL ;
END_VAR
BEGIN
NETWORK
TITLE =
//Ten network celowo jest wolny
NETWORK
TITLE =
// Zapisanie wartosci czasu w pamieci
      A     #STOP;
      FN    #Help_Zbocze_1;
      A     #IN;
      JCN   et_1;
      L     #T_1.PT;
      L     #T_1.ET;
      -D;
      T     #T_1.PT;
      SET;
      R     #T_1.IN;
et_1: NOP   0;
//Przywrocenie czasu zapisanego
      A     #STOP;
      FP    #Help_Zbocze_2;
      A     #IN;
      S     #T_1.IN;
//Warunki poczatkowe
      A     #IN;
      FP    #Help_Zbocze_3;
      A     #STOP;
      JCN   et_3;
      L     #PT;
      T     #T_1.PT;
      SET;
      S     #T_1.IN;
et_3: NOP   0;
//Wywolaj funkcje timera
      CALL  #T_1;
      A     #T_1.Q;
      S     #Q_0;
      AN    #IN;
      A     #STOP;
//Wystaw wyjscie gdy skonczy sie czas
      R     #T_1.IN;
      R     #Q_0;
      L     #T_1.PT;
      L     #T_1.ET;
      -D;
      T     #ET;
//Pokaz wartosc czasu
END_FUNCTION_BLOCK

FUNCTION_BLOCK "T_ON_+_RESET"	// FB 21
//Funkcja zatrzymujaca czas gdy na wejsciu stop pojawi sie stan niski. Wartosc 
//wejscia TON nie jest wtedy brana pod uwage. 
//Dodano przycisk reset.
AUTHOR : Kng
NAME : Help_FB
VERSION : 1.1
VAR_INPUT
  IN : BOOL ;	//Wejscie aktywujace timer
  STOP : BOOL ;	//Sygnal aktywny stanem wysokim
  PT : TIME ;	//Czas zadany
  RESET : BOOL ;	//Wejescie resetujace aktywne stanem wysokim
END_VAR
VAR_OUTPUT
  Q_0 : BOOL ;
END_VAR
VAR_IN_OUT
  ET : TIME ;
END_VAR
VAR
  T_1 : SFB 4;
  Help_Zbocze_1 : BOOL ;
  Help_Zbocze_2 : BOOL ;
  Help_Zbocze_3 : BOOL ;
  Help_Zbocze_4 : BOOL ;
  Help_Zbocze_5 : BOOL ;
END_VAR
BEGIN
NETWORK
TITLE =
//Ten network celowo jest wolny
NETWORK
TITLE =
      A     #RESET;
      S     #Help_Zbocze_4;
// Zapisanie wartosci czasu w pamieci
      A     #STOP;
      FN    #Help_Zbocze_1;
      A     #IN;
      JCN   et_2;
      L     #T_1.PT;
      L     #T_1.ET;
      -D;
      T     #T_1.PT;
      SET;
      R     #T_1.IN;
et_2: NOP   0;
//Przywrocenie czasu zapisanego
      A     #STOP;
      FP    #Help_Zbocze_2;
      A     #IN;
      S     #T_1.IN;
//Wystaw wyjscie gdy skonczy sie czas
      A     #T_1.Q;
      S     #Q_0;
      AN    #IN;
      A     #STOP;
      O;
      A     #RESET;
      R     #T_1.IN;
      R     #Q_0;
//Warunki poczatkowe  oraz reset
      AN    #RESET;
      A     #Help_Zbocze_4;
      O;
      A(;
      A     #IN;
      FP    #Help_Zbocze_3;
      A     #STOP;
      );
      JCN   et_3;
      L     #PT;
      T     #T_1.PT;
      SET;
      R     #Help_Zbocze_4;
//brak wysterownia jezeli reset robiony bez stopu
      A     #STOP;
      S     #T_1.IN;
et_3: NOP   0;
//Wywolaj funkcje timera
      CALL  #T_1;
      L     #T_1.PT;
      L     #T_1.ET;
      -D;
      T     #ET;
//Pokaz wartosc czasu
END_FUNCTION_BLOCK

FUNCTION_BLOCK "Banda_Pojedyncza"	// FB 30
//Funkcja realizujaca koncepcje bandy podwojnej:
//-pojedynczy silnik
//-2 fotokomorki
//
AUTHOR : Kng
FAMILY : Bandy
NAME : B_dual
VERSION : 0.0
VAR_INPUT
  S_Marka_Bezpieczenstwa : BOOL ;
  i_Foto_Koniec : BOOL ;	//Foto na koncu tasmy
  i_Zez_Od_Nast : BOOL ;
  i_Paleta_Dost_Od_Nast : BOOL ;
  i_Zabierz_Od_Pop : BOOL ;
  Czas_Kontroli_Przejazdu : TIME ;
END_VAR
VAR_OUTPUT
  o_Zabierz_Do_Nast : BOOL ;	//Rozkaz pobrania do nast bandy
  o_Zez_Do_Pop : BOOL ;
  o_Paleta_Dost_do_Pop : BOOL ;
  o_Motor_Lewo : BOOL ;
END_VAR
VAR
  Czas_kontrolny : FB 20;
  Help_Motor_Lewo : BOOL ;
  S_Dojazd_Po_Odebraniu : BOOL ;
  S_Help_Zab_Od_Pop : BOOL ;
  Stop_Czas_Kontrolny : BOOL ;
  Zbocze_1 : BOOL ;
  Zbocze_2 : BOOL ;
  Blokada_Wjazd : BOOL ;
  Help_5 : BOOL ;
  Help_6 : BOOL ;
  Help_7 : BOOL ;
  Help_8 : BOOL ;
END_VAR
VAR_TEMP
  Temp_Help_1 : BOOL ;
  Temp_Help_2 : BOOL ;
  Czas_zadany : TIME ;
  Czas_aktualny : TIME ;
END_VAR
BEGIN
NETWORK
TITLE =
//
// B1        B2         foto_1    foto_2         B5        B6
//(\\\\\\\\\\\\\\\\\\)  (\\\\\\\\\\\\\\\\\\)  (\\\\\\\\\\\\\\\\\\)
//                  M1                    M2                     M3
//         
//        zabierz <-- pobierz      |  zabierz    <--  pobierz  
//     zez_do_pop --> zez_od_nast  |  zez_od_pop -->  zez_od_nast
//                                  
//-Uklad dzielony jest na realizowane funkcje
//
//         <----------------------------------------- kierunek
//                  
//
// ten network celowo jest pusty
NETWORK
TITLE =
      A     #S_Marka_Bezpieczenstwa;
      S     #Stop_Czas_Kontrolny;
NETWORK
TITLE =
//Wyznczenie zbocza pozytywnego i negatywnego
//Skocz jezeli brak marki bezpieczenstwa
      AN    #S_Marka_Bezpieczenstwa;
      AN    #Stop_Czas_Kontrolny;
      JC    end;
      AN    #S_Marka_Bezpieczenstwa;
      R     #Stop_Czas_Kontrolny;
NETWORK
TITLE =
// Opis poszczegolnych krokow i skok do nich
// Tasma poprzednia pusta i bierzaca pusta
      AN    #i_Foto_Koniec;
      AN    #o_Zabierz_Do_Nast;
      AN    #Help_Motor_Lewo;
      S     #o_Zez_Do_Pop;
      A     #i_Zabierz_Od_Pop;
      S     #Help_Motor_Lewo;
      S     #Blokada_Wjazd;
//Warunek gdy pobranie z poprzedniej i miejsce foto srodek
//jest zajete
      A     #Help_Motor_Lewo;
      AN    #i_Zabierz_Od_Pop;
      AN    #i_Foto_Koniec;
      =     #Temp_Help_1;
      CALL  #Czas_kontrolny (
           IN                       := #Temp_Help_1,
           STOP                     := #Stop_Czas_Kontrolny,
           PT                       := #Czas_Kontroli_Przejazdu,
           Q_0                      := #Temp_Help_2,
           ET                       := #Czas_aktualny);
//Paleta dostarczona
      A     #Temp_Help_2;
      O;
      A     #i_Foto_Koniec;
      FP    #Zbocze_2;
      R     #Help_Motor_Lewo;
      R     #o_Zez_Do_Pop;
      =     #o_Paleta_Dost_do_Pop;
//jest zezwolenie od nastepnej
      A     #i_Foto_Koniec;
      A     #i_Zez_Od_Nast;
      S     #Help_Motor_Lewo;
      =     #o_Zabierz_Do_Nast;
//Potwierdzenie otrzymania palety
      AN    #Blokada_Wjazd;
      A     #i_Paleta_Dost_Od_Nast;
      FP    #Zbocze_1;
      R     #Help_Motor_Lewo;
//Gdy zajete Foto_1 brak zezwolenia do poprzedniej
      A     #i_Foto_Koniec;
      R     #o_Zez_Do_Pop;
      R     #Blokada_Wjazd;
//warunkowe zakonczenie pracy silnika gdy brak zezwolenia
//z nastepnej
      A     #i_Foto_Koniec;
      AN    #i_Zez_Od_Nast;
      R     #Help_Motor_Lewo;
NETWORK
TITLE =
end:  NOP   0;
      A     #S_Marka_Bezpieczenstwa;
      A     #Help_Motor_Lewo;
      =     #o_Motor_Lewo;
      BEU;
NETWORK
TITLE =
END_FUNCTION_BLOCK

FUNCTION_BLOCK "Banda_Obr_1"	// FB 31
AUTHOR : Kng
FAMILY : Bandy
NAME : Band_obr
VERSION : 0.1
VAR_INPUT
  i_Marka_bezpieczenstwa : BOOL ;
  i_Foto_1 : BOOL ;
  i_Foto_2 : BOOL ;
  i_Zez_od_Nast : BOOL ;
  i_Zabierz_od_Wlot_1 : BOOL ;
  i_Zabierz_od_Wlot_2 : BOOL ;
  i_Paleta_Odb_Wylot : BOOL ;
  i_czuj_poz_Wlot_1 : BOOL ;
  i_czuj_ham_Wlot_1 : BOOL ;
  i_czuj_poz_Wlot_2 : BOOL ;
  i_czuj_ham_Wlot_2 : BOOL ;
  i_Foto_Wlot_1 : BOOL ;
  i_Foto_Wlot_2 : BOOL ;
END_VAR
VAR_OUTPUT
  o_Zez_do_Wlot_1 : BOOL ;
  o_Zez_do_Wlot_2 : BOOL ;
  o_Paleta_Dost_Wlot_1 : BOOL ;
  o_Paleta_Dost_Wlot_2 : BOOL ;
  o_Zabierz_do_Nast : BOOL ;
  o_Motor_1_lewo : BOOL ;
  o_Motor_1_prawo : BOOL ;
  o_Motor_2_obr_s_Wlot_1 : BOOL ;	//Motor obrotnicy,kierunek strona wejscia,szybko
  o_Motor_2_obr_s_Wlot_2 : BOOL ;	//Motor obrotnicy,kierunek strona wyjscia,szybko
  o_Motor_2_Wolno : BOOL ;	//Motor obrotnicy,kierunek strona wejscia,wolno
END_VAR
VAR
  Kontrola_Rolki_Wlot_1 : FB 20;
  Dojazd_Rolki_Wlot_1 : FB 20;
  Kontrola_Rolki_Wlot_2 : FB 20;
  Dojazd_Rolki_Wlot_2 : FB 20;
  Czas_kontrolny : SFB 4;	//Czas kontrolny wjazdu palety
  Sterownie_Obrotnicy : FB 51;
  Opuszczenie_Bandy : SFB 4;
  Silniki_nie_pracuja : BOOL ;
  Help_Motor_1_lewo : BOOL ;
  Help_Motor_1_prawo : BOOL ;
  Help_Motor_2_obr_Wlot_1 : BOOL ;	//Motor obrotnicy,kierunek strona wejscia,szybko
  Help_Motor_2_obr_Wlot_2 : BOOL ;	//Motor obrotnicy,kierunek strona wyjscia,szybko
  Help_Motor_2_Wolno : BOOL ;	//Motor obrotnicy,kierunek strona wejscia,wolno
  Blokada_Na_Wlot_1 : BOOL ;
  Blokada_Na_Wlot_2 : BOOL ;
  Blokada_Wlotu : BOOL ;
  Poz_Wlot_1 : BOOL ;
  Poz_Wlot_2 : BOOL ;
  Obr_Na_Wlot_1 : BOOL ;
  Obr_Na_wlot_2 : BOOL ;
  Odblokuj_Obrotnice : BOOL ;
  Rolki_Odblokowane : BOOL ;
  Stop_Czas_Kontrolny : BOOL ;
  Filtr_Rolki_Wlot_1 : BOOL ;
  H1_Doj_Rolki_Wlot_1 : BOOL ;
  H2_Doj_Rolki_Wlot_1 : BOOL ;
  Filtr_Rolki_Wlot_2 : BOOL ;
  H1_Doj_Rolki_Wlot_2 : BOOL ;
  H2_Doj_Rolki_Wlot_2 : BOOL ;
  Pobranie_Wlot_1 : BOOL ;
  Pobranie_Wlot_2 : BOOL ;
  Paleta_Na_Obrotnicy : BOOL ;
  Oddanie_Palety : BOOL ;
  Zbocze_1 : BOOL ;
  Zbocze_2 : BOOL ;
  Zbocze_3 : BOOL ;
  Wybor_Wjazdu : FB 50;
  Help_Zez_Wlot_1 : BOOL ;
  Help_Zez_Wlot_2 : BOOL ;
END_VAR
VAR_TEMP
  Temp_Help_1 : BOOL ;
  Temp_Help_2 : BOOL ;
  Czas_zadany : TIME ;
  Czas_aktualny : TIME ;
END_VAR
BEGIN
NETWORK
TITLE =
//                   
//Wlot 1                               Wylot
//()()()()|()()()()|  ()()()  |()()()()|()()()()
//()()()()|()()()()| ()()()() |()()()()|()()()()
//()()()()|()()()()| ()()()() |()()()()|()()()()
//()()()()|()()()()| ()()()() |()()()()|()()()()
//()()()()|()()()()|  ()()()  |()()()()|()()()()
//
//                  |()()()()|
//                  |()()()()|
//                  |()()()()| 
//                  |()()()()|
//                    Wlot_2
//         
//          pobierz --> zabierz   |     pobierz --> zabierz   
//     zez_od_nast <-- zez_do_pop | zez_od_nast <-- zez_od_pop
//                                  
//-Uklad dzielony jest na realizowane funkcje
//
//         
//                  
//
// ten network celowo jest pusty
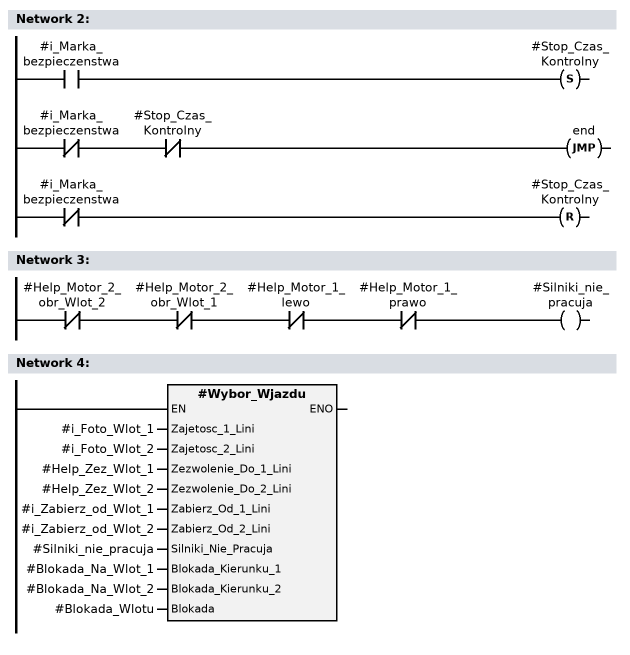
NETWORK
TITLE =
//Zatrzymanie uplywajacego czasu gdy brak bezpieczenstwa
//Skocz jezeli brak marki bezpieczenstwa
      A     #i_Marka_bezpieczenstwa;
      S     #Stop_Czas_Kontrolny;
      AN    #i_Marka_bezpieczenstwa;
      AN    #Stop_Czas_Kontrolny;
      JC    end;
      AN    #i_Marka_bezpieczenstwa;
      R     #Stop_Czas_Kontrolny;
NETWORK
TITLE =
//Sprawdzenie czy silniki nie pracuja
      AN    #Help_Motor_2_obr_Wlot_2;
      AN    #Help_Motor_2_obr_Wlot_1;
      AN    #Help_Motor_1_lewo;
      AN    #Help_Motor_1_prawo;
      =     #Silniki_nie_pracuja;
NETWORK
TITLE =
//Wybranie wjazdu
      CALL  #Wybor_Wjazdu (
           Zajetosc_1_Lini          := #i_Foto_Wlot_1,
           Zajetosc_2_Lini          := #i_Foto_Wlot_2,
           Zezwolenie_Do_1_Lini     := #Help_Zez_Wlot_1,
           Zezwolenie_Do_2_Lini     := #Help_Zez_Wlot_2,
           Zabierz_Od_1_Lini        := #i_Zabierz_od_Wlot_1,
           Zabierz_Od_2_Lini        := #i_Zabierz_od_Wlot_2,
           Silniki_Nie_Pracuja      := #Silniki_nie_pracuja,
           Blokada_Kierunku_1       := #Blokada_Na_Wlot_1,
           Blokada_Kierunku_2       := #Blokada_Na_Wlot_2,
           Blokada                  := #Blokada_Wlotu);
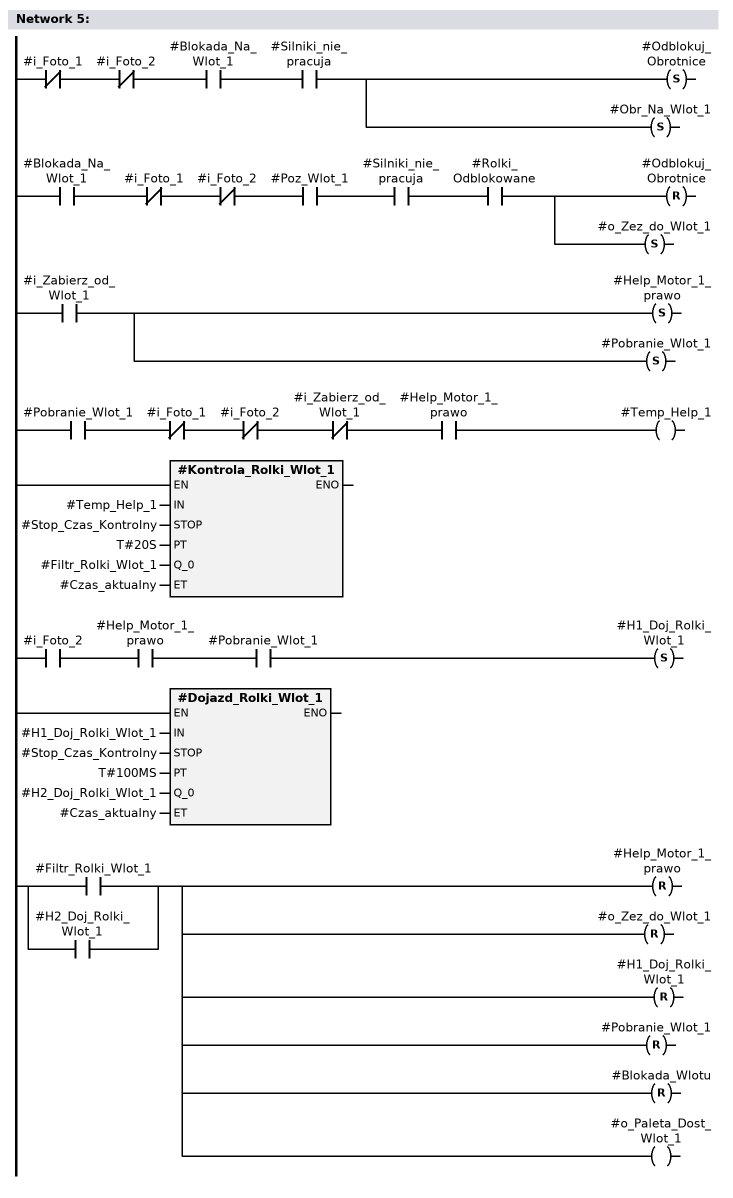
NETWORK
TITLE =
//Pobranie palety z Wlotu nr 1
//Obrot obrotnicy w kierunku wlotu nr 1
      AN    #i_Foto_1;
      AN    #i_Foto_2;
      A     #Blokada_Na_Wlot_1;
      A     #Silniki_nie_pracuja;
      S     #Odblokuj_Obrotnice;
      S     #Obr_Na_Wlot_1;
//Zezwolenie na wjazd z wlotu 1
      A     #Blokada_Na_Wlot_1;
      AN    #i_Foto_1;
      AN    #i_Foto_2;
      A     #Poz_Wlot_1;
      A     #Silniki_nie_pracuja;
      A     #Rolki_Odblokowane;
      R     #Odblokuj_Obrotnice;
      S     #o_Zez_do_Wlot_1;
//Gdy syganl zabierz to uruchom tasme
      A     #i_Zabierz_od_Wlot_1;
      S     #Help_Motor_1_prawo;
      S     #Pobranie_Wlot_1;
//Warunek gdy pobranie z poprzedniej i miejsce foto srodek
//jest zajete
      A     #Pobranie_Wlot_1;
      AN    #i_Foto_1;
      AN    #i_Foto_2;
      AN    #i_Zabierz_od_Wlot_1;
      A     #Help_Motor_1_prawo;
      =     #Temp_Help_1;
      CALL  #Kontrola_Rolki_Wlot_1 (
           IN                       := #Temp_Help_1,
           STOP                     := #Stop_Czas_Kontrolny,
           PT                       := T#20S,
           Q_0                      := #Filtr_Rolki_Wlot_1,
           ET                       := #Czas_aktualny);
      A     #i_Foto_2;
      A     #Help_Motor_1_prawo;
      A     #Pobranie_Wlot_1;
      S     #H1_Doj_Rolki_Wlot_1;
      CALL  #Dojazd_Rolki_Wlot_1 (
           IN                       := #H1_Doj_Rolki_Wlot_1,
           STOP                     := #Stop_Czas_Kontrolny,
           PT                       := T#100MS,
           Q_0                      := #H2_Doj_Rolki_Wlot_1,
           ET                       := #Czas_aktualny);
//Koniec pobierania palety z wlotu 1
      A     #Filtr_Rolki_Wlot_1;
      O;
      A     #H2_Doj_Rolki_Wlot_1;
      R     #Help_Motor_1_prawo;
      R     #o_Zez_do_Wlot_1;
      R     #H1_Doj_Rolki_Wlot_1;
      R     #Pobranie_Wlot_1;
      R     #Blokada_Wlotu;
      =     #o_Paleta_Dost_Wlot_1;
//-----------------------------------------------------
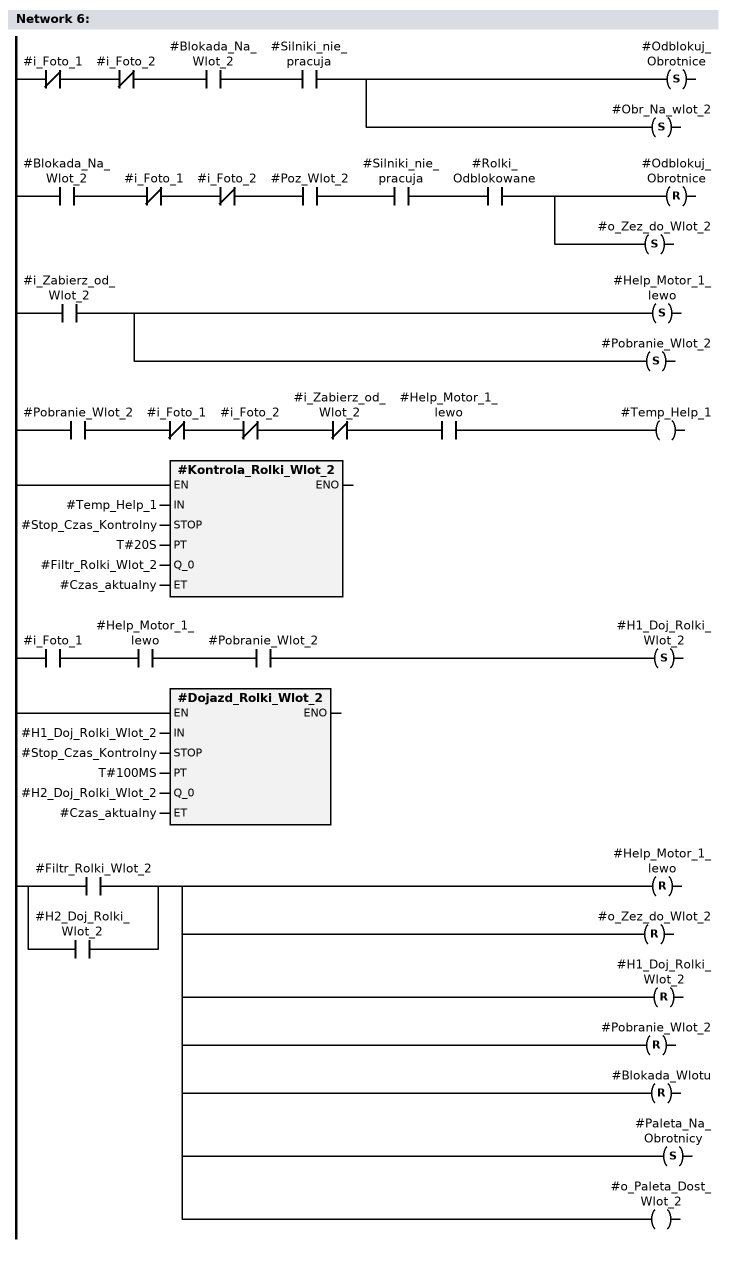
NETWORK
TITLE =
////Pobieranie Palety Wlot 2
//Obrot obrotnicy w kierunku wlotu nr 2
      AN    #i_Foto_1;
      AN    #i_Foto_2;
      A     #Blokada_Na_Wlot_2;
      A     #Silniki_nie_pracuja;
      S     #Odblokuj_Obrotnice;
      S     #Obr_Na_wlot_2;
//Zezwolenie na wjazd z wlotu 2
      A     #Blokada_Na_Wlot_2;
      AN    #i_Foto_1;
      AN    #i_Foto_2;
      A     #Poz_Wlot_2;
      A     #Silniki_nie_pracuja;
      A     #Rolki_Odblokowane;
      R     #Odblokuj_Obrotnice;
      S     #o_Zez_do_Wlot_2;
//Gdy syganl zabierz to uruchom tasme
      A     #i_Zabierz_od_Wlot_2;
      S     #Help_Motor_1_lewo;
      S     #Pobranie_Wlot_2;
//Warunek gdy pobranie z poprzedniej i miejsce foto srodek
//jest zajete
      A     #Pobranie_Wlot_2;
      AN    #i_Foto_1;
      AN    #i_Foto_2;
      AN    #i_Zabierz_od_Wlot_2;
      A     #Help_Motor_1_lewo;
      =     #Temp_Help_1;
      CALL  #Kontrola_Rolki_Wlot_2 (
           IN                       := #Temp_Help_1,
           STOP                     := #Stop_Czas_Kontrolny,
           PT                       := T#20S,
           Q_0                      := #Filtr_Rolki_Wlot_2,
           ET                       := #Czas_aktualny);
      A     #i_Foto_1;
      A     #Help_Motor_1_lewo;
      A     #Pobranie_Wlot_2;
      S     #H1_Doj_Rolki_Wlot_2;
      CALL  #Dojazd_Rolki_Wlot_2 (
           IN                       := #H1_Doj_Rolki_Wlot_2,
           STOP                     := #Stop_Czas_Kontrolny,
           PT                       := T#100MS,
           Q_0                      := #H2_Doj_Rolki_Wlot_2,
           ET                       := #Czas_aktualny);
//Koniec pobierania palety z wlotu 2
      A     #Filtr_Rolki_Wlot_2;
      O;
      A     #H2_Doj_Rolki_Wlot_2;
      R     #Help_Motor_1_lewo;
      R     #o_Zez_do_Wlot_2;
      R     #H1_Doj_Rolki_Wlot_2;
      R     #Pobranie_Wlot_2;
      R     #Blokada_Wlotu;
      S     #Paleta_Na_Obrotnicy;
      =     #o_Paleta_Dost_Wlot_2;
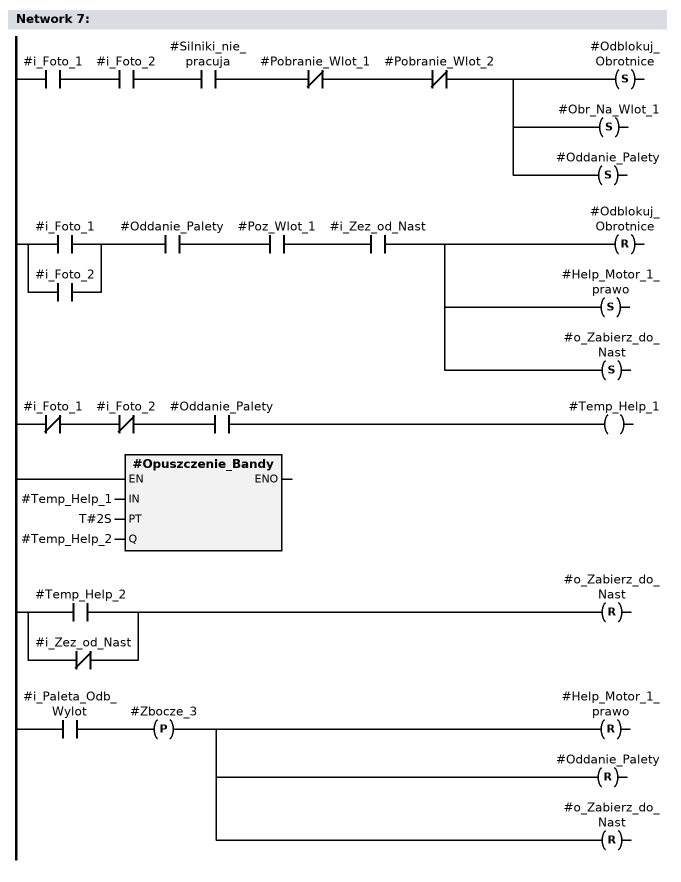
NETWORK
TITLE =
//Wyjazd palety z bandy obrotowej
      A     #i_Foto_1;
      A     #i_Foto_2;
      A     #Silniki_nie_pracuja;
      AN    #Pobranie_Wlot_1;
      AN    #Pobranie_Wlot_2;
      S     #Odblokuj_Obrotnice;
      S     #Obr_Na_Wlot_1;
      S     #Oddanie_Palety;
//Oczekiwanie na zezwolenie
      O     #i_Foto_1;
      O     #i_Foto_2;
      A     #Oddanie_Palety;
      A     #Poz_Wlot_1;
      A     #i_Zez_od_Nast;
      R     #Odblokuj_Obrotnice;
      S     #Help_Motor_1_prawo;
      S     #o_Zabierz_do_Nast;
//reset sygn³u zabierz
      AN    #i_Foto_1;
      AN    #i_Foto_2;
      A     #Oddanie_Palety;
      =     #Temp_Help_1;
      CALL  #Opuszczenie_Bandy (
           IN                       := #Temp_Help_1,
           PT                       := T#2S,
           Q                        := #Temp_Help_2);
      A     #Temp_Help_2;
      O;
      AN    #i_Zez_od_Nast;
      R     #o_Zabierz_do_Nast;
      A     #i_Paleta_Odb_Wylot;
      FP    #Zbocze_3;
      R     #Help_Motor_1_prawo;
      R     #Oddanie_Palety;
      R     #o_Zabierz_do_Nast;
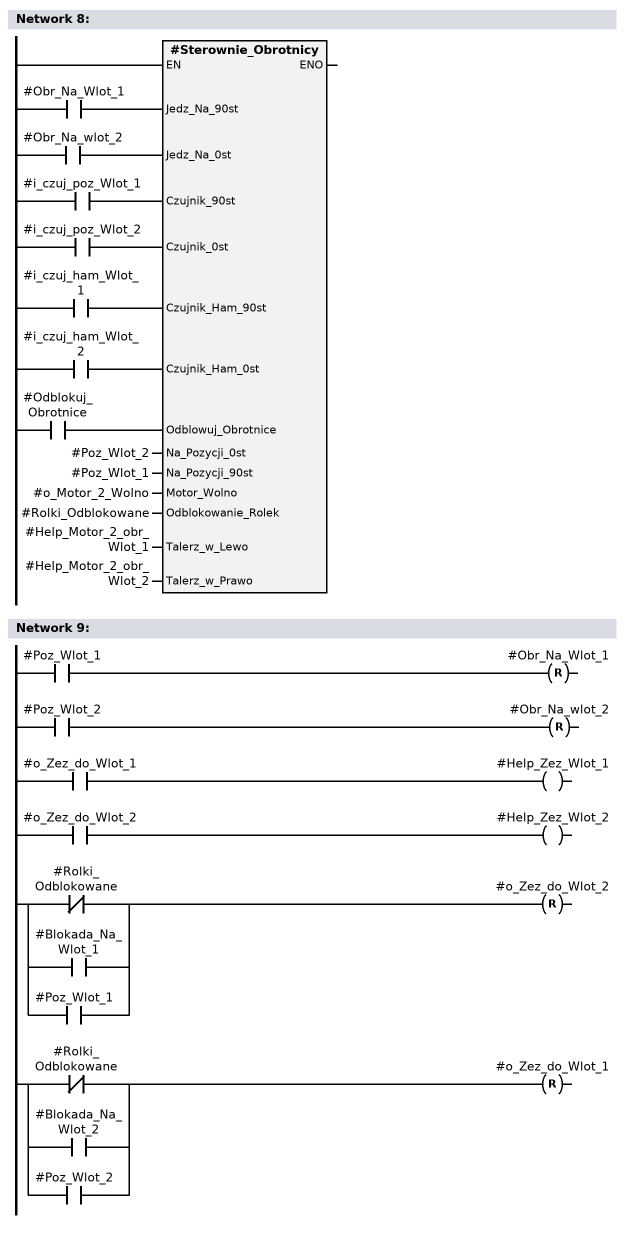
NETWORK
TITLE =
      A     #Obr_Na_Wlot_1;
      =     L 10.0;
      BLD   103;
      A     #Obr_Na_wlot_2;
      =     L 10.1;
      BLD   103;
      A     #i_czuj_poz_Wlot_1;
      =     L 10.2;
      BLD   103;
      A     #i_czuj_poz_Wlot_2;
      =     L 10.3;
      BLD   103;
      A     #i_czuj_ham_Wlot_1;
      =     L 10.4;
      BLD   103;
      A     #i_czuj_ham_Wlot_2;
      =     L 10.5;
      BLD   103;
      A     #Odblokuj_Obrotnice;
      =     L 10.6;
      BLD   103;
      CALL  #Sterownie_Obrotnicy (
           Jedz_Na_90st             := L 10.0,
           Jedz_Na_0st              := L 10.1,
           Czujnik_90st             := L 10.2,
           Czujnik_0st              := L 10.3,
           Czujnik_Ham_90st         := L 10.4,
           Czujnik_Ham_0st          := L 10.5,
           Odblowuj_Obrotnice       := L 10.6,
           Na_Pozycji_0st           := #Poz_Wlot_2,
           Na_Pozycji_90st          := #Poz_Wlot_1,
           Motor_Wolno              := #o_Motor_2_Wolno,
           Odblokowanie_Rolek       := #Rolki_Odblokowane,
           Talerz_w_Lewo            := #Help_Motor_2_obr_Wlot_1,
           Talerz_w_Prawo           := #Help_Motor_2_obr_Wlot_2);
      NOP   0;
NETWORK
TITLE =
//Warunki skrajne
      A     #Poz_Wlot_1;
      R     #Obr_Na_Wlot_1;
      A     #Poz_Wlot_2;
      R     #Obr_Na_wlot_2;
      A     #o_Zez_do_Wlot_1;
      =     #Help_Zez_Wlot_1;
      A     #o_Zez_do_Wlot_2;
      =     #Help_Zez_Wlot_2;
      ON    #Rolki_Odblokowane;
      O     #Blokada_Na_Wlot_1;
      O     #Poz_Wlot_1;
      R     #o_Zez_do_Wlot_2;
      ON    #Rolki_Odblokowane;
      O     #Blokada_Na_Wlot_2;
      O     #Poz_Wlot_2;
      R     #o_Zez_do_Wlot_1;
NETWORK
TITLE =
//Warunki skrajne
end:  NOP   0;
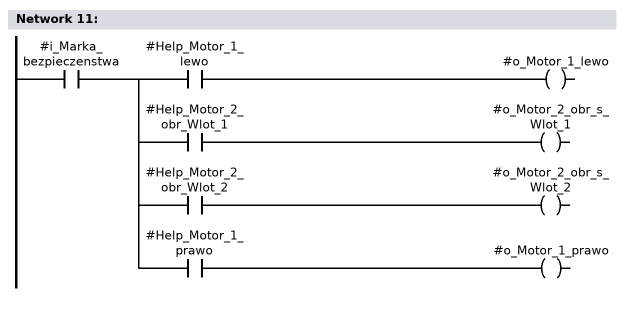
NETWORK
TITLE =
      A     #i_Marka_bezpieczenstwa;
      =     L 10.0;
      A     L 10.0;
      A     #Help_Motor_1_lewo;
      =     #o_Motor_1_lewo;
      A     L 10.0;
      A     #Help_Motor_2_obr_Wlot_1;
      =     #o_Motor_2_obr_s_Wlot_1;
      A     L 10.0;
      A     #Help_Motor_2_obr_Wlot_2;
      =     #o_Motor_2_obr_s_Wlot_2;
      A     L 10.0;
      A     #Help_Motor_1_prawo;
      =     #o_Motor_1_prawo;
NETWORK
TITLE =
END_FUNCTION_BLOCK

FUNCTION_BLOCK "Banda_Obr_2"	// FB 32
AUTHOR : Kng
FAMILY : Bandy
NAME : Band_obr
VERSION : 0.1
VAR_INPUT
  i_Marka_bezpieczenstwa : BOOL ;
  i_Foto_1 : BOOL ;
  i_Foto_2 : BOOL ;
  i_Zez_od_Nast : BOOL ;
  i_Zabierz_od_Wlot_1 : BOOL ;
  i_Zabierz_od_Wlot_2 : BOOL ;
  i_Paleta_Odb_Wylot : BOOL ;
  i_czuj_poz_Wlot_1 : BOOL ;
  i_czuj_ham_Wlot_1 : BOOL ;
  i_czuj_poz_Wlot_2 : BOOL ;
  i_czuj_ham_Wlot_2 : BOOL ;
  i_Czuj_poz_45_deg : BOOL ;
  i_Czuj_ham_45_deg : BOOL ;
  i_Foto_Wlot_1 : BOOL ;
  i_Foto_Wlot_2 : BOOL ;
  i_Etyk_praca_wlacz : BOOL ;
  i_Etyk_poz_podst : BOOL ;
  i_Etyk_obraz_w_pamieci : BOOL ;
  i_Etyk_syg_gotowosci : BOOL ;
  i_Etyk_brak_materialu : BOOL ;
  i_Etyk_Przycisk_Drukuj : BOOL ;
END_VAR
VAR_OUTPUT
  o_Zez_do_Wlot_1 : BOOL ;
  o_Zez_do_Wlot_2 : BOOL ;
  o_Paleta_Dost_Wlot_1 : BOOL ;
  o_Paleta_Dost_Wlot_2 : BOOL ;
  o_Zabierz_do_Nast : BOOL ;
  o_Motor_1_lewo : BOOL ;
  o_Motor_1_prawo : BOOL ;
  o_Motor_2_obr_s_Wlot_1 : BOOL ;	//Motor obrotnicy,kierunek strona wejscia,szybko
  o_Motor_2_obr_s_Wlot_2 : BOOL ;	//Motor obrotnicy,kierunek strona wyjscia,szybko
  o_Motor_2_Wolno : BOOL ;	//Motor obrotnicy,kierunek strona wejscia,wolno
  o_Silownik_etykiety : BOOL ;
  o_Drukuj_Etykiete : BOOL ;
  o_Zalaczenie_Skanera : BOOL ;
  o_Lampka_Przycisk_Drukuj : BOOL ;
END_VAR
VAR
  Kontrola_Rolki_Wlot_1 : FB 20;
  Dojazd_Rolki_Wlot_1 : FB 20;
  Kontrola_Rolki_Wlot_2 : FB 20;
  Dojazd_Rolki_Wlot_2 : FB 20;
  Czas_kontrolny : SFB 4;	//Czas kontrolny wjazdu palety
  Opuszczenie_Bandy : SFB 4;
  Wybor_Wjazdu : FB 50;
  Sterowanie_Obrotu : FB 52;
  Czas_Oczek_Na_Obraz : SFB 4;
  Silniki_nie_pracuja : BOOL ;
  Help_Motor_1_lewo : BOOL ;
  Help_Motor_1_prawo : BOOL ;
  Help_Motor_2_obr_Wlot_1 : BOOL ;	//Motor obrotnicy,kierunek strona wejscia,szybko
  Help_Motor_2_obr_Wlot_2 : BOOL ;	//Motor obrotnicy,kierunek strona wyjscia,szybko
  Help_Motor_2_Wolno : BOOL ;	//Motor obrotnicy,kierunek strona wejscia,wolno
  Blokada_Na_Wlot_1 : BOOL ;
  Blokada_Na_Wlot_2 : BOOL ;
  Blokada_Wlotu : BOOL ;
  Poz_Wlot_1 : BOOL ;
  Poz_Wlot_2 : BOOL ;
  Obr_Na_Wlot_1 : BOOL ;
  Obr_Na_wlot_2 : BOOL ;
  Odblokuj_Obrotnice : BOOL ;
  Rolki_Odblokowane : BOOL ;
  Stop_Czas_Kontrolny : BOOL ;
  Filtr_Rolki_Wlot_1 : BOOL ;
  H1_Doj_Rolki_Wlot_1 : BOOL ;
  H2_Doj_Rolki_Wlot_1 : BOOL ;
  Filtr_Rolki_Wlot_2 : BOOL ;
  H1_Doj_Rolki_Wlot_2 : BOOL ;
  H2_Doj_Rolki_Wlot_2 : BOOL ;
  Pobranie_Wlot_1 : BOOL ;
  Pobranie_Wlot_2 : BOOL ;
  Paleta_Na_Obrotnicy : BOOL ;
  Oddanie_Palety : BOOL ;
  Help_Zez_Wlot_1 : BOOL ;
  Help_Zez_Wlot_2 : BOOL ;
  Obr_Na_Etykieciarke : BOOL ;
  Poz_Etykieciarka : BOOL ;
  Help_Silownik_Etyk : BOOL ;
  Oczekiwanie_Na_Obraz : BOOL ;
  Help_ety_przykl : BOOL ;
  Zbocze_przecisku_drukuj : BOOL ;
  Sprawdzenie_Etyk : BOOL ;
  Zbocze_1 : BOOL ;
  Zbocze_2 : BOOL ;
  Zbocze_3 : BOOL ;
  Zbocze_4 : BOOL ;
  H1 : BOOL ;
  H2 : BOOL ;
  H3 : BOOL ;
  H4 : BOOL ;
  H5 : BOOL ;
  H6 : BOOL ;
  H7 : BOOL ;
END_VAR
VAR_TEMP
  Temp_Help_1 : BOOL ;
  Temp_Help_2 : BOOL ;
  Czas_zadany : TIME ;
  Czas_aktualny : TIME ;
END_VAR
BEGIN
NETWORK
TITLE =
//                   
//Wlot 1                               Wylot
//()()()()|()()()()|  ()()()  |()()()()|()()()()
//()()()()|()()()()| ()()()() |()()()()|()()()()
//()()()()|()()()()| ()()()() |()()()()|()()()()
//()()()()|()()()()| ()()()() |()()()()|()()()()
//()()()()|()()()()|  ()()()  |()()()()|()()()()
//
//                  |()()()()|
//                  |()()()()|
//                  |()()()()| 
//                  |()()()()|
//                    Wlot_2
//         
//          pobierz --> zabierz   |     pobierz --> zabierz   
//     zez_od_nast <-- zez_do_pop | zez_od_nast <-- zez_od_pop
//                                  
//-Uklad dzielony jest na realizowane funkcje
//
//         
//                  
//
// ten network celowo jest pusty
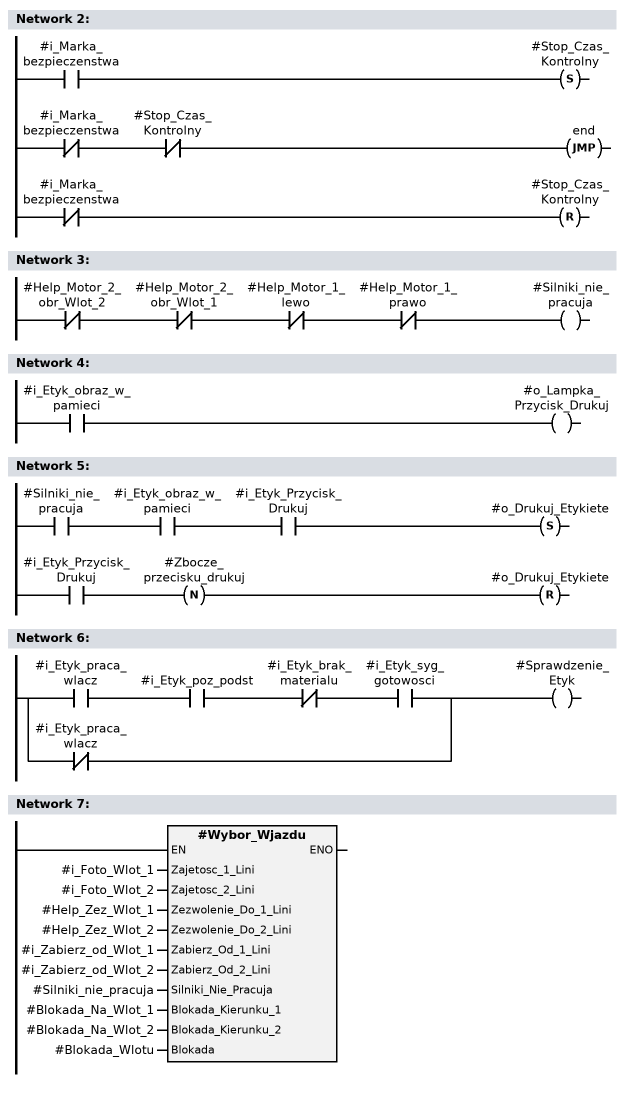
NETWORK
TITLE =
//Zatrzymanie uplywajacego czasu gdy brak bezpieczenstwa
//Skocz jezeli brak marki bezpieczenstwa
      A     #i_Marka_bezpieczenstwa;
      S     #Stop_Czas_Kontrolny;
      AN    #i_Marka_bezpieczenstwa;
      AN    #Stop_Czas_Kontrolny;
      JC    end;
      AN    #i_Marka_bezpieczenstwa;
      R     #Stop_Czas_Kontrolny;
NETWORK
TITLE =
//Sprawdzenie czy silniki nie pracuja
      AN    #Help_Motor_2_obr_Wlot_2;
      AN    #Help_Motor_2_obr_Wlot_1;
      AN    #Help_Motor_1_lewo;
      AN    #Help_Motor_1_prawo;
      =     #Silniki_nie_pracuja;
NETWORK
TITLE =
      A     #i_Etyk_obraz_w_pamieci;
      =     #o_Lampka_Przycisk_Drukuj;
NETWORK
TITLE =
//Drukowanie samej etykiety
      A     #Silniki_nie_pracuja;
      A     #i_Etyk_obraz_w_pamieci;
      A     #i_Etyk_Przycisk_Drukuj;
      S     #o_Drukuj_Etykiete;
      A     #i_Etyk_Przycisk_Drukuj;
      FN    #Zbocze_przecisku_drukuj;
      R     #o_Drukuj_Etykiete;
      NOP   0;
NETWORK
TITLE =
//Sprawdzenie etykietownicy zanim pobrana paleta
//Warunki pobrania palety gdy praca z etykietami
      A     #i_Etyk_praca_wlacz;
      A     #i_Etyk_poz_podst;
      AN    #i_Etyk_brak_materialu;	// gdy brak materialu
      A     #i_Etyk_syg_gotowosci;
      ON    #i_Etyk_praca_wlacz;
      =     #Sprawdzenie_Etyk;
NETWORK
TITLE =
//Wybranie wjazdu
      CALL  #Wybor_Wjazdu (
           Zajetosc_1_Lini          := #i_Foto_Wlot_1,
           Zajetosc_2_Lini          := #i_Foto_Wlot_2,
           Zezwolenie_Do_1_Lini     := #Help_Zez_Wlot_1,
           Zezwolenie_Do_2_Lini     := #Help_Zez_Wlot_2,
           Zabierz_Od_1_Lini        := #i_Zabierz_od_Wlot_1,
           Zabierz_Od_2_Lini        := #i_Zabierz_od_Wlot_2,
           Silniki_Nie_Pracuja      := #Silniki_nie_pracuja,
           Blokada_Kierunku_1       := #Blokada_Na_Wlot_1,
           Blokada_Kierunku_2       := #Blokada_Na_Wlot_2,
           Blokada                  := #Blokada_Wlotu);
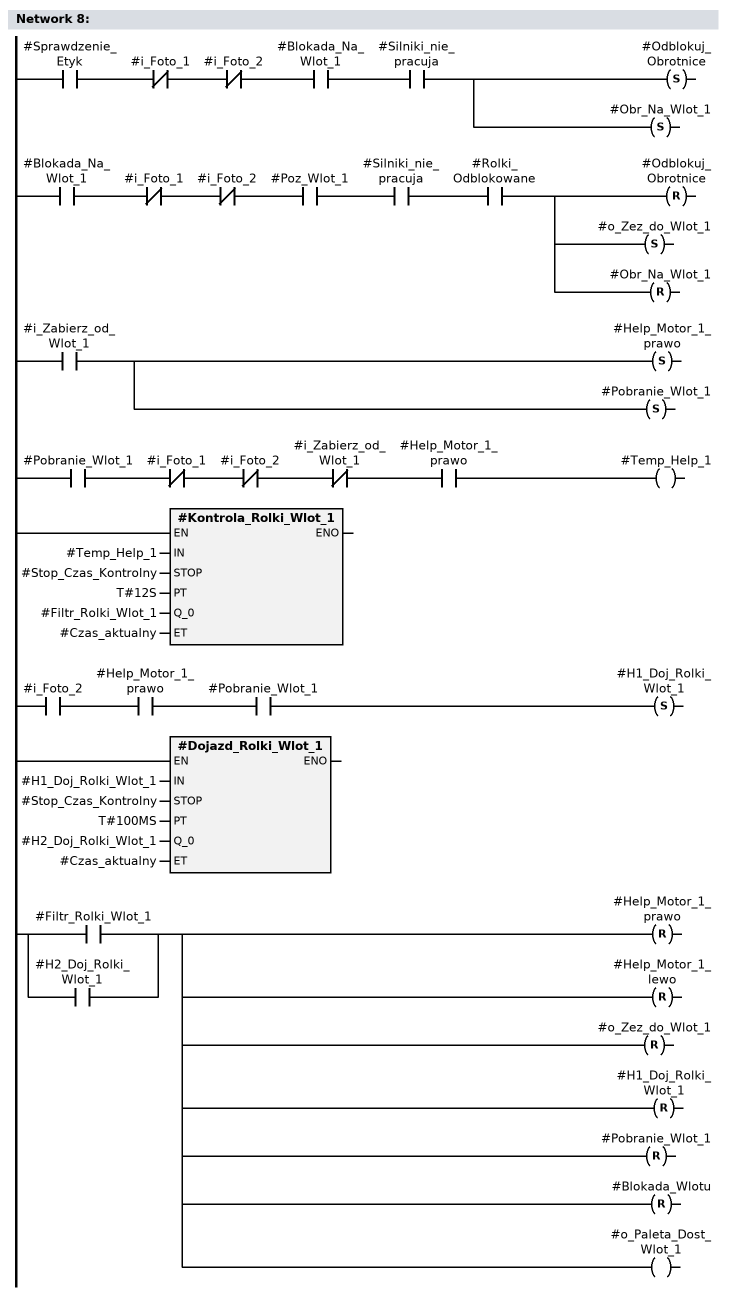
NETWORK
TITLE =
//Pobranie palety z Wlotu nr 1
//Obrot obrotnicy w kierunku wlotu nr 1
      A     #Sprawdzenie_Etyk;
      AN    #i_Foto_1;
      AN    #i_Foto_2;
      A     #Blokada_Na_Wlot_1;
      A     #Silniki_nie_pracuja;
      S     #Odblokuj_Obrotnice;
      S     #Obr_Na_Wlot_1;
//Zezwolenie na wjazd z wlotu 1
      A     #Blokada_Na_Wlot_1;
      AN    #i_Foto_1;
      AN    #i_Foto_2;
      A     #Poz_Wlot_1;
      A     #Silniki_nie_pracuja;
      A     #Rolki_Odblokowane;
      R     #Odblokuj_Obrotnice;
      S     #o_Zez_do_Wlot_1;
      R     #Obr_Na_Wlot_1;
//Gdy syganl zabierz to uruchom tasme
      A     #i_Zabierz_od_Wlot_1;
      S     #Help_Motor_1_prawo;
      S     #Pobranie_Wlot_1;
//Warunek gdy pobranie z poprzedniej i miejsce foto srodek
//jest zajete
      A     #Pobranie_Wlot_1;
      AN    #i_Foto_1;
      AN    #i_Foto_2;
      AN    #i_Zabierz_od_Wlot_1;
      A     #Help_Motor_1_prawo;
      =     #Temp_Help_1;
      CALL  #Kontrola_Rolki_Wlot_1 (
           IN                       := #Temp_Help_1,
           STOP                     := #Stop_Czas_Kontrolny,
           PT                       := T#12S,
           Q_0                      := #Filtr_Rolki_Wlot_1,
           ET                       := #Czas_aktualny);
      A     #i_Foto_2;
      A     #Help_Motor_1_prawo;
      A     #Pobranie_Wlot_1;
      S     #H1_Doj_Rolki_Wlot_1;
      CALL  #Dojazd_Rolki_Wlot_1 (
           IN                       := #H1_Doj_Rolki_Wlot_1,
           STOP                     := #Stop_Czas_Kontrolny,
           PT                       := T#100MS,
           Q_0                      := #H2_Doj_Rolki_Wlot_1,
           ET                       := #Czas_aktualny);
//Koniec pobierania palety z wlotu 1
      A     #Filtr_Rolki_Wlot_1;
      O;
      A     #H2_Doj_Rolki_Wlot_1;
      R     #Help_Motor_1_prawo;
      R     #Help_Motor_1_lewo;
      R     #o_Zez_do_Wlot_1;
      R     #H1_Doj_Rolki_Wlot_1;
      R     #Pobranie_Wlot_1;
      R     #Blokada_Wlotu;
      =     #o_Paleta_Dost_Wlot_1;
//-----------------------------------------------------
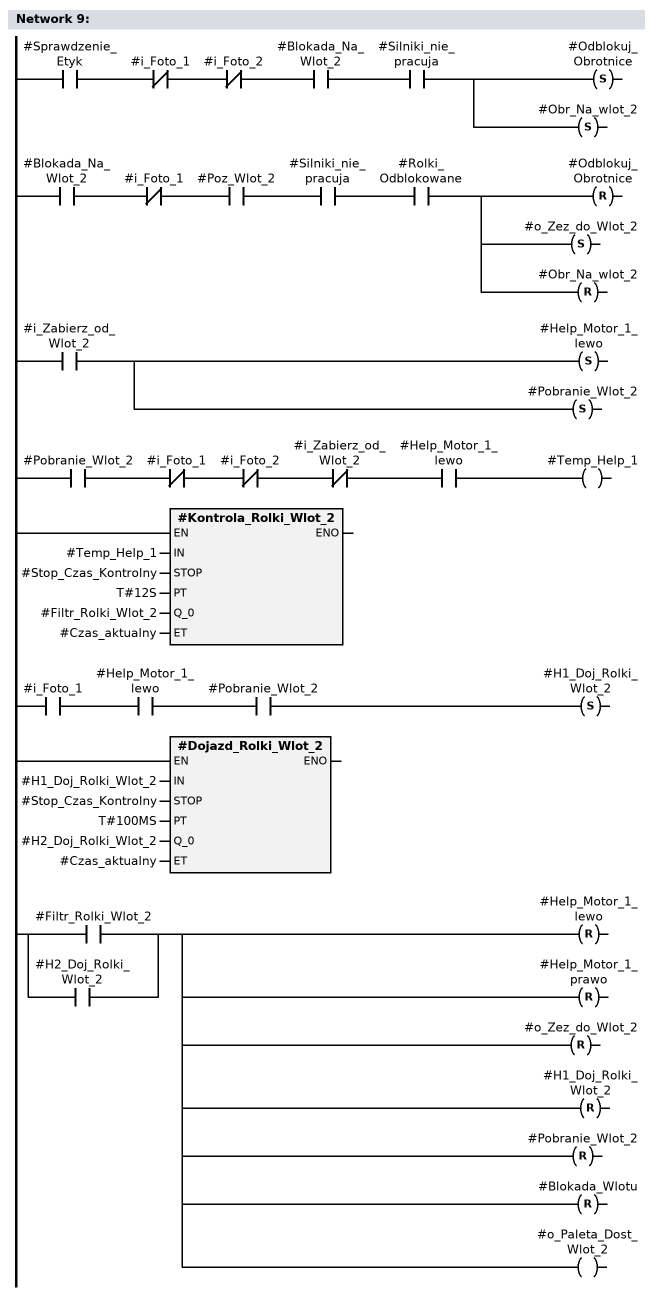
NETWORK
TITLE =
////Pobieranie Palety Wlot 2
//Obrot obrotnicy w kierunku wlotu nr 2
      A     #Sprawdzenie_Etyk;
      AN    #i_Foto_1;
      AN    #i_Foto_2;
      A     #Blokada_Na_Wlot_2;
      A     #Silniki_nie_pracuja;
      S     #Odblokuj_Obrotnice;
      S     #Obr_Na_wlot_2;
//Zezwolenie na wjazd z wlotu 2
      A     #Blokada_Na_Wlot_2;
      AN    #i_Foto_1;
      A     #Poz_Wlot_2;
      A     #Silniki_nie_pracuja;
      A     #Rolki_Odblokowane;
      R     #Odblokuj_Obrotnice;
      S     #o_Zez_do_Wlot_2;
      R     #Obr_Na_wlot_2;
//Gdy syganl zabierz to uruchom tasme
      A     #i_Zabierz_od_Wlot_2;
      S     #Help_Motor_1_lewo;
      S     #Pobranie_Wlot_2;
//Warunek gdy pobranie z poprzedniej i miejsce foto srodek
//jest zajete
      A     #Pobranie_Wlot_2;
      AN    #i_Foto_1;
      AN    #i_Foto_2;
      AN    #i_Zabierz_od_Wlot_2;
      A     #Help_Motor_1_lewo;
      =     #Temp_Help_1;
      CALL  #Kontrola_Rolki_Wlot_2 (
           IN                       := #Temp_Help_1,
           STOP                     := #Stop_Czas_Kontrolny,
           PT                       := T#12S,
           Q_0                      := #Filtr_Rolki_Wlot_2,
           ET                       := #Czas_aktualny);
      A     #i_Foto_1;
      A     #Help_Motor_1_lewo;
      A     #Pobranie_Wlot_2;
      S     #H1_Doj_Rolki_Wlot_2;
      CALL  #Dojazd_Rolki_Wlot_2 (
           IN                       := #H1_Doj_Rolki_Wlot_2,
           STOP                     := #Stop_Czas_Kontrolny,
           PT                       := T#100MS,
           Q_0                      := #H2_Doj_Rolki_Wlot_2,
           ET                       := #Czas_aktualny);
//Koniec pobierania palety z wlotu 2
      A     #Filtr_Rolki_Wlot_2;
      O;
      A     #H2_Doj_Rolki_Wlot_2;
      R     #Help_Motor_1_lewo;
      R     #Help_Motor_1_prawo;
      R     #o_Zez_do_Wlot_2;
      R     #H1_Doj_Rolki_Wlot_2;
      R     #Pobranie_Wlot_2;
      R     #Blokada_Wlotu;
      =     #o_Paleta_Dost_Wlot_2;
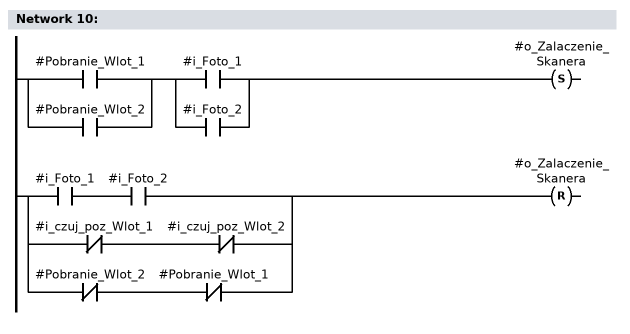
NETWORK
TITLE =
//Zalczenie skanera etykiet
      A(;
      O     #Pobranie_Wlot_1;
      O     #Pobranie_Wlot_2;
      );
      A(;
      O     #i_Foto_1;
      O     #i_Foto_2;
      );
      S     #o_Zalaczenie_Skanera;
      A(;
      A     #i_Foto_1;
      A     #i_Foto_2;
      O;
      AN    #i_czuj_poz_Wlot_1;
      AN    #i_czuj_poz_Wlot_2;
      O;
      AN    #Pobranie_Wlot_2;
      AN    #Pobranie_Wlot_1;
      );
      R     #o_Zalaczenie_Skanera;
      NOP   0;
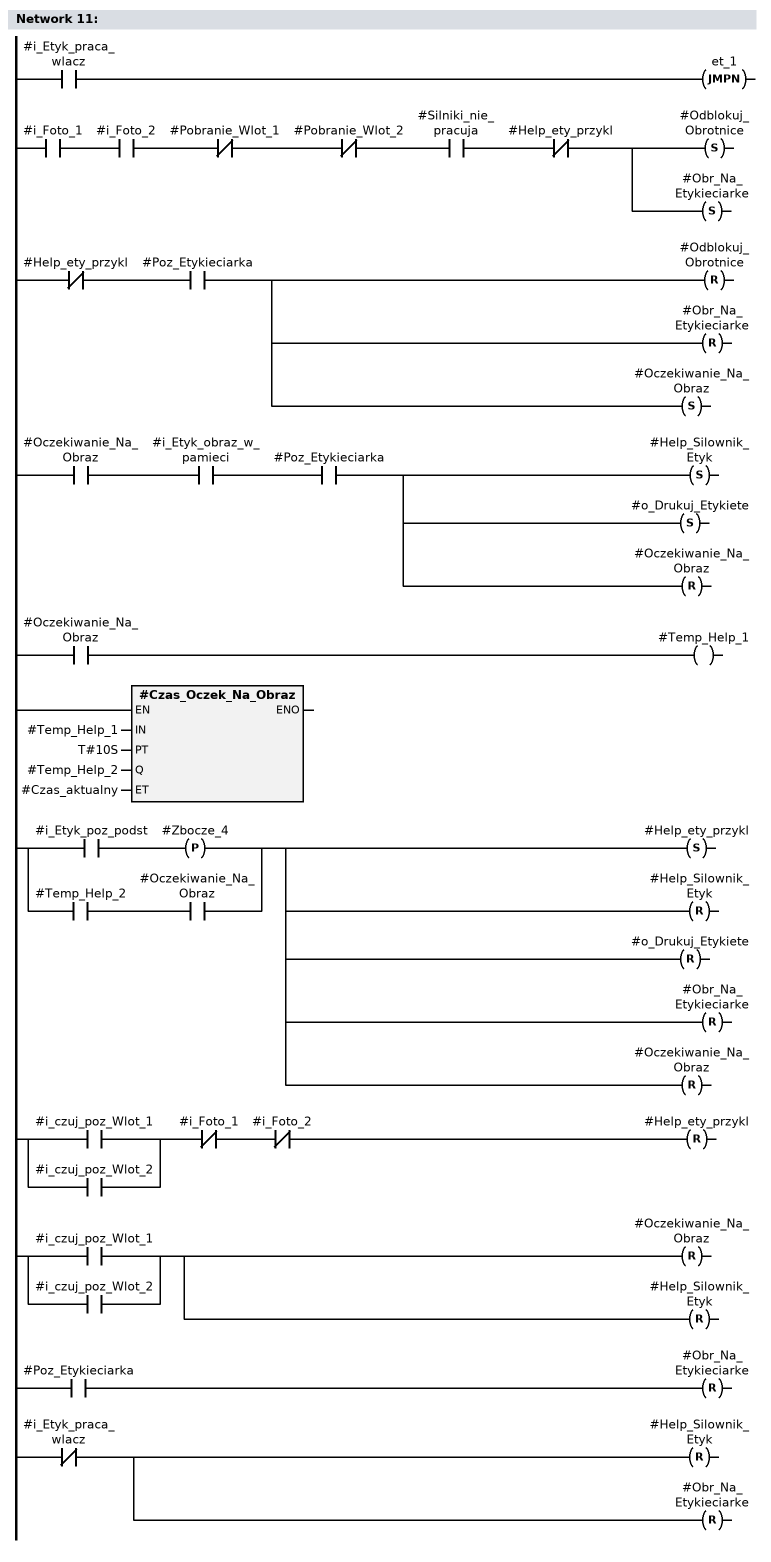
NETWORK
TITLE =
//Dojazd palety na etykieciarke
//Praca z etykietowaniem
      A     #i_Etyk_praca_wlacz;
      JCN   et_1;
// Obrot palety na maszyne etykietujaca
      A     #i_Foto_1;
      A     #i_Foto_2;
      AN    #Pobranie_Wlot_1;
      AN    #Pobranie_Wlot_2;
      A     #Silniki_nie_pracuja;
      AN    #Help_ety_przykl;
      S     #Odblokuj_Obrotnice;
      S     #Obr_Na_Etykieciarke;
//Oczekiwanie na
      AN    #Help_ety_przykl;
      A     #Poz_Etykieciarka;
      R     #Odblokuj_Obrotnice;
      R     #Obr_Na_Etykieciarke;
      S     #Oczekiwanie_Na_Obraz;
//Czas wstrzymania az obraz dotrze do etykieciarki
      A     #Oczekiwanie_Na_Obraz;
      A     #i_Etyk_obraz_w_pamieci;
      A     #Poz_Etykieciarka;	//dopisano 14.05.2014
      S     #Help_Silownik_Etyk;
      S     #o_Drukuj_Etykiete;
      R     #Oczekiwanie_Na_Obraz;
//Czas kontrolny oczekiwania na obraz
      A     #Oczekiwanie_Na_Obraz;
      =     #Temp_Help_1;
      CALL  #Czas_Oczek_Na_Obraz (
           IN                       := #Temp_Help_1,
           PT                       := T#10S,
           Q                        := #Temp_Help_2,
           ET                       := #Czas_aktualny);
//zakonczenie przyklejania etykiety
      A     #i_Etyk_poz_podst;
      FP    #Zbocze_4;
      O;
      A     #Temp_Help_2;
      A     #Oczekiwanie_Na_Obraz;
      S     #Help_ety_przykl;
      R     #Help_Silownik_Etyk;
      R     #o_Drukuj_Etykiete;
      R     #Obr_Na_Etykieciarke;
      R     #Oczekiwanie_Na_Obraz;	//dopisano 14.05.2014
//Warunkowy reset bitu przyklejania etykiety  
et_1: NOP   0;
      O     #i_czuj_poz_Wlot_1;
      O     #i_czuj_poz_Wlot_2;
      AN    #i_Foto_1;
      AN    #i_Foto_2;
      R     #Help_ety_przykl;
      O     #i_czuj_poz_Wlot_1;
      O     #i_czuj_poz_Wlot_2;
      R     #Oczekiwanie_Na_Obraz;
      R     #Help_Silownik_Etyk;
      A     #Poz_Etykieciarka;
      R     #Obr_Na_Etykieciarke;
      AN    #i_Etyk_praca_wlacz;
      R     #Help_Silownik_Etyk;
      R     #Obr_Na_Etykieciarke;
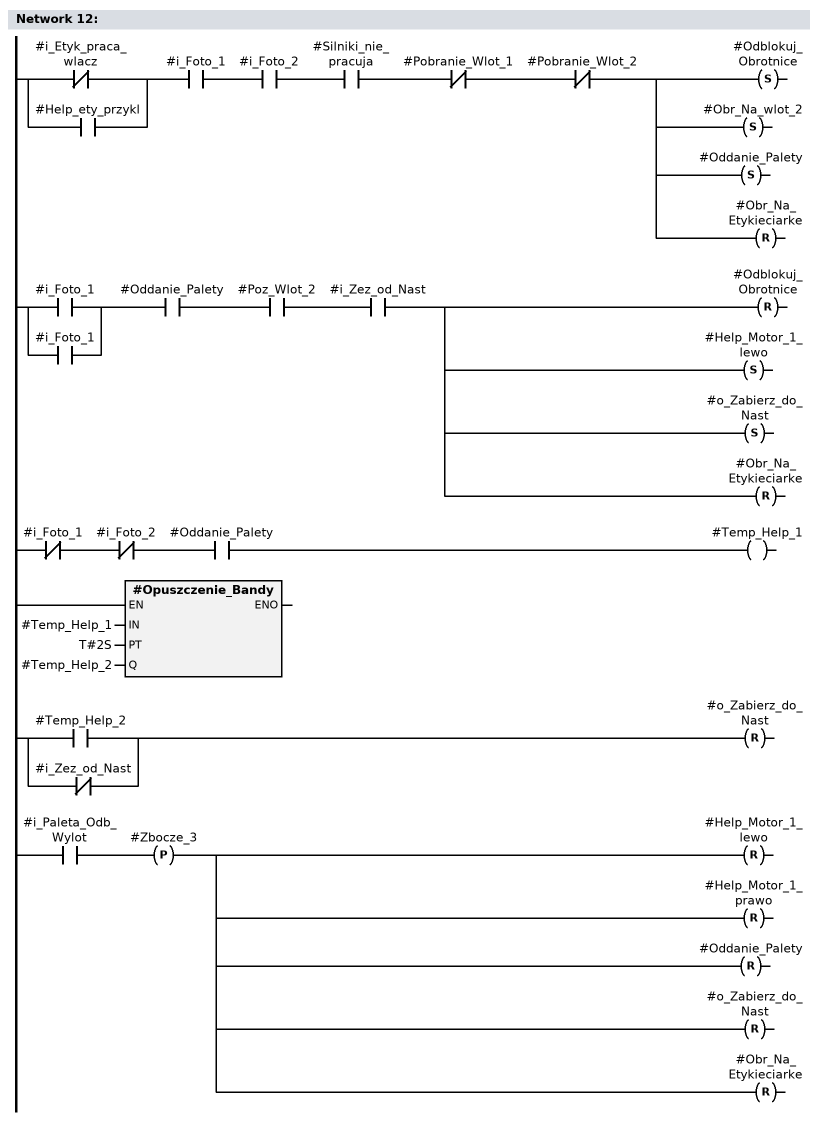
NETWORK
TITLE =
//Wyjazd palety z bandy obrotowej
//Jazda w kierunku wylotu
      ON    #i_Etyk_praca_wlacz;
      O     #Help_ety_przykl;
      A(;
      A     #i_Foto_1;
      A     #i_Foto_2;
      A     #Silniki_nie_pracuja;
      AN    #Pobranie_Wlot_1;
      AN    #Pobranie_Wlot_2;
      );
      S     #Odblokuj_Obrotnice;
      S     #Obr_Na_wlot_2;
      S     #Oddanie_Palety;
      R     #Obr_Na_Etykieciarke;
//Oczekiwanie na zezwolenie
      O     #i_Foto_1;
      O     #i_Foto_1;
      A     #Oddanie_Palety;
      A     #Poz_Wlot_2;
      A     #i_Zez_od_Nast;
      R     #Odblokuj_Obrotnice;
      S     #Help_Motor_1_lewo;
      S     #o_Zabierz_do_Nast;
      R     #Obr_Na_Etykieciarke;
//reset sygnalu zabierz
      AN    #i_Foto_1;
      AN    #i_Foto_2;
      A     #Oddanie_Palety;
      =     #Temp_Help_1;
      CALL  #Opuszczenie_Bandy (
           IN                       := #Temp_Help_1,
           PT                       := T#2S,
           Q                        := #Temp_Help_2);
      A     #Temp_Help_2;
      O;
      AN    #i_Zez_od_Nast;
      R     #o_Zabierz_do_Nast;
      A     #i_Paleta_Odb_Wylot;
//Otrzymanie sygalu zwrotnego o odbiorze palety
      FP    #Zbocze_3;
      R     #Help_Motor_1_lewo;
      R     #Help_Motor_1_prawo;
      R     #Oddanie_Palety;
      R     #o_Zabierz_do_Nast;
      R     #Obr_Na_Etykieciarke;
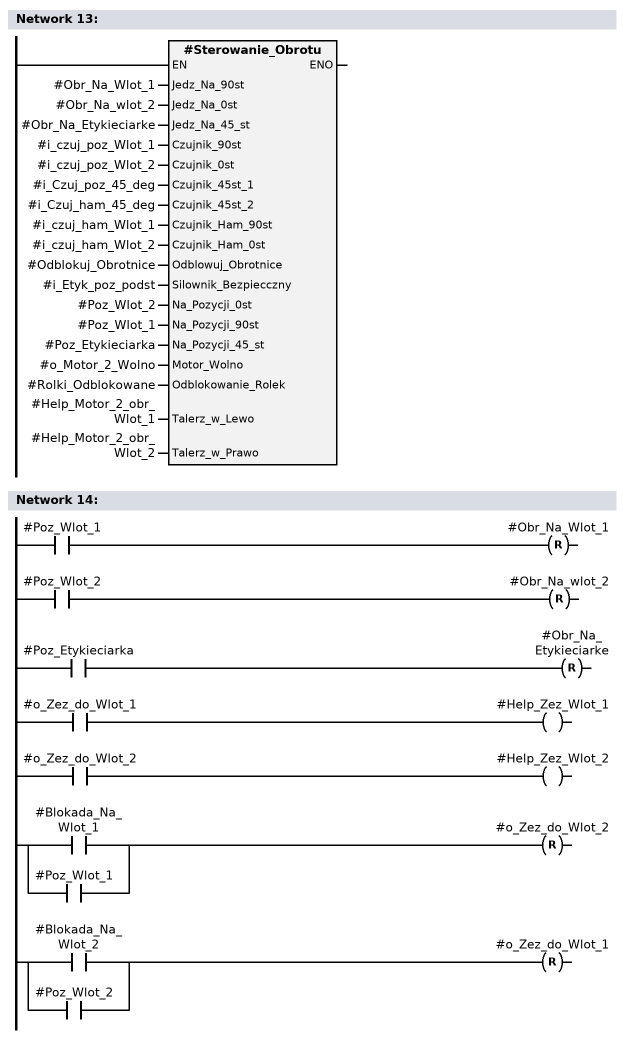
NETWORK
TITLE =
//Obrot na pozycje 
      CALL  #Sterowanie_Obrotu (
           Jedz_Na_90st             := #Obr_Na_Wlot_1,
           Jedz_Na_0st              := #Obr_Na_wlot_2,
           Jedz_Na_45_st            := #Obr_Na_Etykieciarke,
           Czujnik_90st             := #i_czuj_poz_Wlot_1,
           Czujnik_0st              := #i_czuj_poz_Wlot_2,
           Czujnik_45st_1           := #i_Czuj_poz_45_deg,
           Czujnik_45st_2           := #i_Czuj_ham_45_deg,
           Czujnik_Ham_90st         := #i_czuj_ham_Wlot_1,
           Czujnik_Ham_0st          := #i_czuj_ham_Wlot_2,
           Odblowuj_Obrotnice       := #Odblokuj_Obrotnice,
           Silownik_Bezpiecczny     := #i_Etyk_poz_podst,
           Na_Pozycji_0st           := #Poz_Wlot_2,
           Na_Pozycji_90st          := #Poz_Wlot_1,
           Na_Pozycji_45_st         := #Poz_Etykieciarka,
           Motor_Wolno              := #o_Motor_2_Wolno,
           Odblokowanie_Rolek       := #Rolki_Odblokowane,
           Talerz_w_Lewo            := #Help_Motor_2_obr_Wlot_1,
           Talerz_w_Prawo           := #Help_Motor_2_obr_Wlot_2);
NETWORK
TITLE =
//Warunki skrajne
      A     #Poz_Wlot_1;
      R     #Obr_Na_Wlot_1;
      A     #Poz_Wlot_2;
      R     #Obr_Na_wlot_2;
      A     #Poz_Etykieciarka;
      R     #Obr_Na_Etykieciarke;
      A     #o_Zez_do_Wlot_1;
      =     #Help_Zez_Wlot_1;
      A     #o_Zez_do_Wlot_2;
      =     #Help_Zez_Wlot_2;
      O     #Blokada_Na_Wlot_1;
      O     #Poz_Wlot_1;
      R     #o_Zez_do_Wlot_2;
      O     #Blokada_Na_Wlot_2;
      O     #Poz_Wlot_2;
      R     #o_Zez_do_Wlot_1;
NETWORK
TITLE =
//Warunki skrajne
end:  NOP   0;
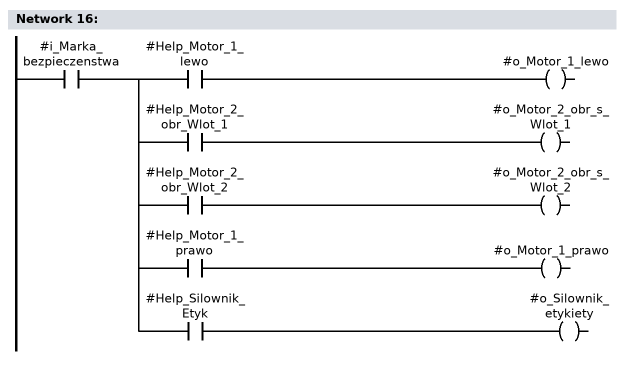
NETWORK
TITLE =
      A     #i_Marka_bezpieczenstwa;
      =     L 10.0;
      A     L 10.0;
      A     #Help_Motor_1_lewo;
      =     #o_Motor_1_lewo;
      A     L 10.0;
      A     #Help_Motor_2_obr_Wlot_1;
      =     #o_Motor_2_obr_s_Wlot_1;
      A     L 10.0;
      A     #Help_Motor_2_obr_Wlot_2;
      =     #o_Motor_2_obr_s_Wlot_2;
      A     L 10.0;
      A     #Help_Motor_1_prawo;
      =     #o_Motor_1_prawo;
      A     L 10.0;
      A     #Help_Silownik_Etyk;
      =     #o_Silownik_etykiety;
NETWORK
TITLE =
END_FUNCTION_BLOCK

